LIN {X -109.277,Y -17.308,Z -54.438,A -90.000,B 90.000,C 0.000} C_DIS
LIN {X -109.528,Y -17.308,Z -53.967,A -90.000,B 90.000,C 0.000} C_DIS
LIN {X -109.760,Y -17.308,Z -53.459,A -90.000,B 90.000,C 0.000} C_DIS
LIN {X -109.870,Y -17.308,Z -53.202,A -90.000,B 90.000,C 0.000} C_DIS
LIN {X -109.990,Y -17.308,Z -52.935,A -90.000,B 90.000,C 0.000} C_DIS
LIN {X -110.022,Y -17.308,Z -52.850,A -90.000,B 90.000,C 0.000} C_DIS
LIN {X -110.260,Y -17.308,Z -52.116,A -90.000,B 90.000,C 0.000} C_DIS
LIN {X -110.354,Y -17.308,Z -51.704,A -90.000,B 90.000,C 0.000} C_DIS
LIN {X -110.399,Y -17.308,Z -51.283,A -90.000,B 90.000,C 0.000} C_DIS
LIN {X -110.450,Y -17.308,Z -50.683,A -90.000,B 90.000,C 0.000} C_DIS
LIN {X -110.444,Y -17.308,Z -50.213,A -90.000,B 90.000,C 0.000} C_DIS
LIN {X -110.434,Y -17.308,Z -50.113,A -90.000,B 90.000,C 0.000} C_DIS
LIN {X -110.392,Y -17.308,Z -49.798,A -90.000,B 90.000,C 0.000} C_DIS
LIN {X -110.361,Y -17.308,Z -49.609,A -90.000,B 90.000,C 0.000} C_DIS
LIN {X -110.302,Y -17.308,Z -49.301,A -90.000,B 90.000,C 0.000} C_DIS
LIN {X -110.171,Y -17.308,Z -48.794,A -90.000,B 90.000,C 0.000} C_DIS
LIN {X -110.038,Y -17.308,Z -48.429,A -90.000,B 90.000,C 0.000} C_DIS
LIN {X -109.863,Y -17.308,Z -47.985,A -90.000,B 90.000,C 0.000} C_DIS
LIN {X -109.731,Y -17.308,Z -47.725,A -90.000,B 90.000,C 0.000} C_DIS
LIN {X -109.686,Y -17.308,Z -47.627,A -90.000,B 90.000,C 0.000} C_DIS
LIN {X -109.488,Y -17.308,Z -47.252,A -90.000,B 90.000,C 0.000} C_DIS
LIN {X -109.413,Y -17.308,Z -47.127,A -90.000,B 90.000,C 0.000} C_DIS
LIN {X -109.830,Y -17.308,Z -46.394,A -90.000,B 90.000,C 0.000} C_DIS
LIN {X -109.928,Y -17.308,Z -46.209,A -90.000,B 90.000,C 0.000} C_DIS
LIN {X -110.117,Y -17.308,Z -45.841,A -90.000,B 90.000,C 0.000} C_DIS
LIN {X -110.455,Y -17.308,Z -45.092,A -90.000,B 90.000,C 0.000} C_DIS
LIN {X -110.509,Y -17.308,Z -44.961,A -90.000,B 90.000,C 0.000} C_DIS
LIN {X -110.701,Y -17.308,Z -44.445,A -90.000,B 90.000,C 0.000} C_DIS
LIN {X -110.791,Y -17.308,Z -44.174,A -90.000,B 90.000,C 0.000} C_DIS
LIN {X -110.988,Y -17.308,Z -43.576,A -90.000,B 90.000,C 0.000} C_DIS
LIN {X -111.093,Y -17.308,Z -43.162,A -90.000,B 90.000,C 0.000} C_DIS
LIN {X -111.179,Y -17.308,Z -42.781,A -90.000,B 90.000,C 0.000} C_DIS
LIN {X -111.225,Y -17.308,Z -42.559,A -90.000,B 90.000,C 0.000} C_DIS
LIN {X -111.305,Y -17.308,Z -42.009,A -90.000,B 90.000,C 0.000} C_DIS
LIN {X -111.349,Y -17.308,Z -41.588,A -90.000,B 90.000,C 0.000} C_DIS
LIN {X -111.368,Y -17.308,Z -41.241,A -90.000,B 90.000,C 0.000} C_DIS
LIN {X -111.364,Y -17.308,Z -40.978,A -90.000,B 90.000,C 0.000} C_DIS
LIN {X -111.359,Y -17.308,Z -40.623,A -90.000,B 90.000,C 0.000} C_DIS
LIN {X -111.346,Y -17.308,Z -40.304,A -90.000,B 90.000,C 0.000} C_DIS
LIN {X -111.305,Y -17.308,Z -39.903,A -90.000,B 90.000,C 0.000} C_DIS
LIN {X -111.262,Y -17.308,Z -39.606,A -90.000,B 90.000,C 0.000} C_DIS
LIN {X -111.171,Y -17.308,Z -39.214,A -90.000,B 90.000,C 0.000} C_DIS
LIN {X -111.102,Y -17.308,Z -38.934,A -90.000,B 90.000,C 0.000} C_DIS
LIN {X -110.936,Y -17.308,Z -38.436,A -90.000,B 90.000,C 0.000} C_DIS
LIN {X -110.874,Y -17.308,Z -38.268,A -90.000,B 90.000,C 0.000} C_DIS
LIN {X -110.765,Y -17.308,Z -38.003,A -90.000,B 90.000,C 0.000} C_DIS
LIN {X -110.667,Y -17.308,Z -37.794,A -90.000,B 90.000,C 0.000} C_DIS
LIN {X -110.600,Y -17.308,Z -37.663,A -90.000,B 90.000,C 0.000} C_DIS
LIN {X -110.459,Y -17.308,Z -37.399,A -90.000,B 90.000,C 0.000} C_DIS
LIN {X -110.237,Y -17.308,Z -37.056,A -90.000,B 90.000,C 0.000} C_DIS
LIN {X -110.078,Y -17.308,Z -36.846,A -90.000,B 90.000,C 0.000} C_DIS
LIN {X -109.834,Y -17.308,Z -36.557,A -90.000,B 90.000,C 0.000} C_DIS
LIN {X -109.557,Y -17.308,Z -36.304,A -90.000,B 90.000,C 0.000} C_DIS
LIN {X -109.328,Y -17.308,Z -36.101,A -90.000,B 90.000,C 0.000} C_DIS
LIN {X -109.011,Y -17.308,Z -35.882,A -90.000,B 90.000,C 0.000} C_DIS
LIN {X -108.744,Y -17.308,Z -35.735,A -90.000,B 90.000,C 0.000} C_DIS
LIN {X -108.407,Y -17.308,Z -35.562,A -90.000,B 90.000,C 0.000} C_DIS
LIN {X -108.370,Y -17.308,Z -35.547,A -90.000,B 90.000,C 0.000} C_DIS
LIN {X -108.101,Y -17.308,Z -35.424,A -90.000,B 90.000,C 0.000} C_DIS
LIN {X -108.024,Y -17.308,Z -35.397,A -90.000,B 90.000,C 0.000} C_DIS
LIN {X -107.986,Y -17.308,Z -35.382,A -90.000,B 90.000,C 0.000} C_DIS
LIN {X -107.790,Y -17.308,Z -35.138,A -90.000,B 90.000,C 0.000} C_DIS
LIN {X -107.687,Y -17.308,Z -35.003,A -90.000,B 90.000,C 0.000} C_DIS
LIN {X -107.576,Y -17.308,Z -34.852,A -90.000,B 90.000,C 0.000} C_DIS
LIN {X -107.363,Y -17.308,Z -34.573,A -90.000,B 90.000,C 0.000} C_DIS
LIN {X -107.172,Y -17.308,Z -34.351,A -90.000,B 90.000,C 0.000} C_DIS
LIN {X -106.994,Y -17.308,Z -34.130,A -90.000,B 90.000,C 0.000} C_DIS
LIN {X -106.743,Y -17.308,Z -33.884,A -90.000,B 90.000,C 0.000} C_DIS
LIN {X -106.465,Y -17.308,Z -33.618,A -90.000,B 90.000,C 0.000} C_DIS
LIN {X -106.295,Y -17.308,Z -33.457,A -90.000,B 90.000,C 0.000} C_DIS
LIN {X -105.896,Y -17.308,Z -33.133,A -90.000,B 90.000,C 0.000} C_DIS
LIN {X -105.714,Y -17.308,Z -32.987,A -90.000,B 90.000,C 0.000} C_DIS
LIN {X -104.978,Y -17.308,Z -32.450,A -90.000,B 90.000,C 0.000} C_DIS
LIN {X -104.425,Y -17.308,Z -32.079,A -90.000,B 90.000,C 0.000} C_DIS
LIN {X -104.048,Y -17.308,Z -31.825,A -90.000,B 90.000,C 0.000} C_DIS
LIN {X -103.908,Y -17.308,Z -31.733,A -90.000,B 90.000,C 0.000} C_DIS
LIN {X -103.388,Y -17.308,Z -31.409,A -90.000,B 90.000,C 0.000} C_DIS
LIN {X -102.835,Y -17.308,Z -31.110,A -90.000,B 90.000,C 0.000} C_DIS
LIN {X -102.526,Y -17.308,Z -30.944,A -90.000,B 90.000,C 0.000} C_DIS
LIN {X -102.329,Y -17.308,Z -30.848,A -90.000,B 90.000,C 0.000} C_DIS
LIN {X -101.877,Y -17.308,Z -30.649,A -90.000,B 90.000,C 0.000} C_DIS
LIN {X -101.633,Y -17.308,Z -30.551,A -90.000,B 90.000,C 0.000} C_DIS
LIN {X -101.290,Y -17.308,Z -30.421,A -90.000,B 90.000,C 0.000} C_DIS
LIN {X -100.896,Y -17.308,Z -30.282,A -90.000,B 90.000,C 0.000} C_DIS
LIN {X -100.530,Y -17.308,Z -30.139,A -90.000,B 90.000,C 0.000} C_DIS
LIN {X -100.458,Y -17.308,Z -29.896,A -90.000,B 90.000,C 0.000} C_DIS
LIN {X -100.322,Y -17.308,Z -29.499,A -90.000,B 90.000,C 0.000} C_DIS
LIN {X -100.161,Y -17.308,Z -29.156,A -90.000,B 90.000,C 0.000} C_DIS
LIN {X -99.930,Y -17.308,Z -28.698,A -90.000,B 90.000,C 0.000} C_DIS
LIN {X -99.695,Y -17.308,Z -28.324,A -90.000,B 90.000,C 0.000} C_DIS
LIN {X -99.528,Y -17.308,Z -28.064,A -90.000,B 90.000,C 0.000} C_DIS
LIN {X -99.432,Y -17.308,Z -27.919,A -90.000,B 90.000,C 0.000} C_DIS
LIN {X -99.092,Y -17.308,Z -27.475,A -90.000,B 90.000,C 0.000} C_DIS
LIN {X -98.825,Y -17.308,Z -27.155,A -90.000,B 90.000,C 0.000} C_DIS
LIN {X -98.539,Y -17.308,Z -26.819,A -90.000,B 90.000,C 0.000} C_DIS
LIN {X -98.265,Y -17.308,Z -26.515,A -90.000,B 90.000,C 0.000} C_DIS
LIN {X -98.055,Y -17.308,Z -26.298,A -90.000,B 90.000,C 0.000} C_DIS
LIN {X -97.848,Y -17.308,Z -26.093,A -90.000,B 90.000,C 0.000} C_DIS
LIN {X -97.651,Y -17.308,Z -25.907,A -90.000,B 90.000,C 0.000} C_DIS
LIN {X -97.470,Y -17.308,Z -25.741,A -90.000,B 90.000,C 0.000} C_DIS
LIN {X -97.372,Y -17.308,Z -25.646,A -90.000,B 90.000,C 0.000} C_DIS
LIN {X -97.070,Y -17.308,Z -25.379,A -90.000,B 90.000,C 0.000} C_DIS
LIN {X -96.977,Y -17.308,Z -25.311,A -90.000,B 90.000,C 0.000} C_DIS
LIN {X -96.877,Y -17.308,Z -25.234,A -90.000,B 90.000,C 0.000} C_DIS
LIN {X -96.544,Y -17.308,Z -25.007,A -90.000,B 90.000,C 0.000} C_DIS
LIN {X -96.186,Y -17.308,Z -24.822,A -90.000,B 90.000,C 0.000} C_DIS
LIN {X -95.601,Y -17.308,Z -24.606,A -90.000,B 90.000,C 0.000} C_DIS
LIN {X -95.394,Y -17.308,Z -24.551,A -90.000,B 90.000,C 0.000} C_DIS
LIN {X -95.167,Y -17.308,Z -24.498,A -90.000,B 90.000,C 0.000} C_DIS
LIN {X -95.084,Y -17.308,Z -24.484,A -90.000,B 90.000,C 0.000} C_DIS
LIN {X -94.665,Y -17.308,Z -24.424,A -90.000,B 90.000,C 0.000} C_DIS
LIN {X -94.242,Y -17.308,Z -24.415,A -90.000,B 90.000,C 0.000} C_DIS
LIN {X -94.028,Y -17.308,Z -24.425,A -90.000,B 90.000,C 0.000} C_DIS
LIN {X -93.391,Y -17.308,Z -24.450,A -90.000,B 90.000,C 0.000} C_DIS
LIN {X -93.076,Y -17.308,Z -24.495,A -90.000,B 90.000,C 0.000} C_DIS
LIN {X -92.696,Y -17.308,Z -24.538,A -90.000,B 90.000,C 0.000} C_DIS
LIN {X -92.367,Y -17.308,Z -24.604,A -90.000,B 90.000,C 0.000} C_DIS
LIN {X -92.079,Y -17.308,Z -24.636,A -90.000,B 90.000,C 0.000} C_DIS
LIN {X -91.937,Y -17.308,Z -24.654,A -90.000,B 90.000,C 0.000} C_DIS
LIN {X -91.341,Y -17.308,Z -24.709,A -90.000,B 90.000,C 0.000} C_DIS
LIN {X -90.954,Y -17.308,Z -24.728,A -90.000,B 90.000,C 0.000} C_DIS
LIN {X -90.765,Y -17.308,Z -24.739,A -90.000,B 90.000,C 0.000} C_DIS
LIN {X -90.252,Y -17.308,Z -24.737,A -90.000,B 90.000,C 0.000} C_DIS
LIN {X -89.583,Y -17.308,Z -24.703,A -90.000,B 90.000,C 0.000} C_DIS
LIN {X -89.336,Y -17.308,Z -24.674,A -90.000,B 90.000,C 0.000} C_DIS
LIN {X -88.613,Y -17.308,Z -24.546,A -90.000,B 90.000,C 0.000} C_DIS
LIN {X -88.432,Y -17.308,Z -24.502,A -90.000,B 90.000,C 0.000} C_DIS
LIN {X -88.062,Y -17.308,Z -24.386,A -90.000,B 90.000,C 0.000} C_DIS
LIN {X -87.996,Y -17.308,Z -24.360,A -90.000,B 90.000,C 0.000} C_DIS
LIN {X -87.766,Y -17.308,Z -24.270,A -90.000,B 90.000,C 0.000} C_DIS
LIN {X -87.464,Y -17.308,Z -24.122,A -90.000,B 90.000,C 0.000} C_DIS
LIN {X -87.249,Y -17.308,Z -23.989,A -90.000,B 90.000,C 0.000} C_DIS
LIN {X -87.134,Y -17.308,Z -23.898,A -90.000,B 90.000,C 0.000} C_DIS
LIN {X -87.088,Y -17.308,Z -23.852,A -90.000,B 90.000,C 0.000} C_DIS
LIN {X -86.793,Y -17.308,Z -23.483,A -90.000,B 90.000,C 0.000} C_DIS
LIN {X -86.245,Y -17.308,Z -22.709,A -90.000,B 90.000,C 0.000} C_DIS
LIN {X -85.958,Y -17.308,Z -22.315,A -90.000,B 90.000,C 0.000} C_DIS
LIN {X -85.762,Y -17.308,Z -22.052,A -90.000,B 90.000,C 0.000} C_DIS
LIN {X -85.514,Y -17.308,Z -21.715,A -90.000,B 90.000,C 0.000} C_DIS
LIN {X -85.447,Y -17.308,Z -21.614,A -90.000,B 90.000,C 0.000} C_DIS
LIN {X -85.429,Y -17.308,Z -21.548,A -90.000,B 90.000,C 0.000} C_DIS
LIN {X -85.386,Y -17.308,Z -21.370,A -90.000,B 90.000,C 0.000} C_DIS
LIN {X -85.352,Y -17.308,Z -21.224,A -90.000,B 90.000,C 0.000} C_DIS
LIN {X -85.295,Y -17.308,Z -21.008,A -90.000,B 90.000,C 0.000} C_DIS
LIN {X -85.173,Y -17.308,Z -20.564,A -90.000,B 90.000,C 0.000} C_DIS
LIN {X -85.006,Y -17.308,Z -20.118,A -90.000,B 90.000,C 0.000} C_DIS
LIN {X -84.875,Y -17.308,Z -19.788,A -90.000,B 90.000,C 0.000} C_DIS
LIN {X -84.669,Y -17.308,Z -19.377,A -90.000,B 90.000,C 0.000} C_DIS
LIN {X -84.438,Y -17.308,Z -18.974,A -90.000,B 90.000,C 0.000} C_DIS
LIN {X -84.069,Y -17.308,Z -18.464,A -90.000,B 90.000,C 0.000} C_DIS
LIN {X -83.972,Y -17.308,Z -18.336,A -90.000,B 90.000,C 0.000} C_DIS
LIN {X -83.659,Y -17.308,Z -17.989,A -90.000,B 90.000,C 0.000} C_DIS
LIN {X -83.310,Y -17.308,Z -17.678,A -90.000,B 90.000,C 0.000} C_DIS
LIN {X -83.039,Y -17.308,Z -17.445,A -90.000,B 90.000,C 0.000} C_DIS
LIN {X -82.804,Y -17.308,Z -17.264,A -90.000,B 90.000,C 0.000} C_DIS
LIN {X -82.421,Y -17.308,Z -17.018,A -90.000,B 90.000,C 0.000} C_DIS
LIN {X -82.064,Y -17.308,Z -16.803,A -90.000,B 90.000,C 0.000} C_DIS
LIN {X -81.656,Y -17.308,Z -16.601,A -90.000,B 90.000,C 0.000} C_DIS
LIN {X -81.272,Y -17.308,Z -16.447,A -90.000,B 90.000,C 0.000} C_DIS
LIN {X -80.773,Y -17.308,Z -16.264,A -90.000,B 90.000,C 0.000} C_DIS
LIN {X -80.331,Y -17.308,Z -16.156,A -90.000,B 90.000,C 0.000} C_DIS
LIN {X -79.940,Y -17.308,Z -16.064,A -90.000,B 90.000,C 0.000} C_DIS
LIN {X -79.763,Y -17.308,Z -16.028,A -90.000,B 90.000,C 0.000} C_DIS
LIN {X -79.312,Y -17.308,Z -15.968,A -90.000,B 90.000,C 0.000} C_DIS
LIN {X -78.986,Y -17.308,Z -15.938,A -90.000,B 90.000,C 0.000} C_DIS
LIN {X -78.616,Y -17.308,Z -15.911,A -90.000,B 90.000,C 0.000} C_DIS
LIN {X -78.161,Y -17.308,Z -15.902,A -90.000,B 90.000,C 0.000} C_DIS
LIN {X -77.499,Y -17.308,Z -15.925,A -90.000,B 90.000,C 0.000} C_DIS
LIN {X -77.301,Y -17.308,Z -15.936,A -90.000,B 90.000,C 0.000} C_DIS
LIN {X -76.909,Y -17.308,Z -15.971,A -90.000,B 90.000,C 0.000} C_DIS
LIN {X -76.875,Y -17.308,Z -15.976,A -90.000,B 90.000,C 0.000} C_DIS
LIN {X -75.728,Y -17.308,Z -16.188,A -90.000,B 90.000,C 0.000} C_DIS
LIN {X -75.480,Y -17.308,Z -16.245,A -90.000,B 90.000,C 0.000} C_DIS
LIN {X -74.439,Y -17.308,Z -16.560,A -90.000,B 90.000,C 0.000} C_DIS
LIN {X -73.971,Y -17.308,Z -16.709,A -90.000,B 90.000,C 0.000} C_DIS
LIN {X -72.559,Y -17.308,Z -17.306,A -90.000,B 90.000,C 0.000} C_DIS
LIN {X -72.171,Y -17.308,Z -17.515,A -90.000,B 90.000,C 0.000} C_DIS
LIN {X -71.532,Y -17.308,Z -17.863,A -90.000,B 90.000,C 0.000} C_DIS
LIN {X -71.248,Y -17.308,Z -18.011,A -90.000,B 90.000,C 0.000} C_DIS
LIN {X -70.853,Y -17.308,Z -18.223,A -90.000,B 90.000,C 0.000} C_DIS
LIN {X -70.304,Y -17.308,Z -18.552,A -90.000,B 90.000,C 0.000} C_DIS
LIN {X -69.506,Y -17.308,Z -19.020,A -90.000,B 90.000,C 0.000} C_DIS
LIN {X -69.055,Y -17.308,Z -19.311,A -90.000,B 90.000,C 0.000} C_DIS
LIN {X -67.940,Y -17.308,Z -20.084,A -90.000,B 90.000,C 0.000} C_DIS
LIN {X -67.668,Y -17.308,Z -20.290,A -90.000,B 90.000,C 0.000} C_DIS
LIN {X -67.045,Y -17.308,Z -20.777,A -90.000,B 90.000,C 0.000} C_DIS
LIN {X -66.717,Y -17.308,Z -21.045,A -90.000,B 90.000,C 0.000} C_DIS
LIN {X -66.444,Y -17.308,Z -21.276,A -90.000,B 90.000,C 0.000} C_DIS
LIN {X -65.961,Y -17.308,Z -21.696,A -90.000,B 90.000,C 0.000} C_DIS
LIN {X -65.767,Y -17.308,Z -21.893,A -90.000,B 90.000,C 0.000} C_DIS
LIN {X -65.312,Y -17.308,Z -22.358,A -90.000,B 90.000,C 0.000} C_DIS
LIN {X -64.845,Y -17.308,Z -22.810,A -90.000,B 90.000,C 0.000} C_DIS
LIN {X -64.258,Y -17.308,Z -23.509,A -90.000,B 90.000,C 0.000} C_DIS
LIN {X -63.904,Y -17.308,Z -23.932,A -90.000,B 90.000,C 0.000} C_DIS
LIN {X -63.462,Y -17.308,Z -24.494,A -90.000,B 90.000,C 0.000} C_DIS
LIN {X -63.348,Y -17.308,Z -24.652,A -90.000,B 90.000,C 0.000} C_DIS
LIN {X -63.215,Y -17.308,Z -24.848,A -90.000,B 90.000,C 0.000} C_DIS
LIN {X -62.785,Y -17.308,Z -25.397,A -90.000,B 90.000,C 0.000} C_DIS
LIN {X -62.557,Y -17.308,Z -25.702,A -90.000,B 90.000,C 0.000} C_DIS
LIN {X -62.483,Y -17.308,Z -25.777,A -90.000,B 90.000,C 0.000} C_DIS
LIN {X -62.054,Y -17.308,Z -26.201,A -90.000,B 90.000,C 0.000} C_DIS
LIN {X -61.340,Y -17.308,Z -26.673,A -90.000,B 90.000,C 0.000} C_DIS
LIN {X -60.531,Y -17.308,Z -27.025,A -90.000,B 90.000,C 0.000} C_DIS
LIN {X -60.319,Y -17.308,Z -27.118,A -90.000,B 90.000,C 0.000} C_DIS
LIN {X -58.849,Y -17.308,Z -27.587,A -90.000,B 90.000,C 0.000} C_DIS
LIN {X -56.852,Y -17.308,Z -28.118,A -90.000,B 90.000,C 0.000} C_DIS
LIN {X -56.644,Y -17.308,Z -28.164,A -90.000,B 90.000,C 0.000} C_DIS
LIN {X -55.206,Y -17.308,Z -28.534,A -90.000,B 90.000,C 0.000} C_DIS
LIN {X -54.599,Y -17.308,Z -28.678,A -90.000,B 90.000,C 0.000} C_DIS
LIN {X -53.961,Y -17.308,Z -28.823,A -90.000,B 90.000,C 0.000} C_DIS
LIN {X -52.713,Y -17.308,Z -29.052,A -90.000,B 90.000,C 0.000} C_DIS
LIN {X -52.238,Y -17.308,Z -29.158,A -90.000,B 90.000,C 0.000} C_DIS
LIN {X -50.712,Y -17.308,Z -29.450,A -90.000,B 90.000,C 0.000} C_DIS
LIN {X -49.140,Y -17.308,Z -29.676,A -90.000,B 90.000,C 0.000} C_DIS
LIN {X -48.828,Y -17.308,Z -29.708,A -90.000,B 90.000,C 0.000} C_DIS
LIN {X -45.658,Y -17.308,Z -30.077,A -90.000,B 90.000,C 0.000} C_DIS
LIN {X -45.116,Y -17.308,Z -30.119,A -90.000,B 90.000,C 0.000} C_DIS
LIN {X -44.038,Y -17.308,Z -30.215,A -90.000,B 90.000,C 0.000} C_DIS
LIN {X -41.956,Y -17.308,Z -30.414,A -90.000,B 90.000,C 0.000} C_DIS
LIN {X -40.163,Y -17.308,Z -30.556,A -90.000,B 90.000,C 0.000} C_DIS
LIN {X -39.196,Y -17.308,Z -30.672,A -90.000,B 90.000,C 0.000} C_DIS
LIN {X -36.171,Y -17.308,Z -31.051,A -90.000,B 90.000,C 0.000} C_DIS
LIN {X -34.413,Y -17.308,Z -31.305,A -90.000,B 90.000,C 0.000} C_DIS
LIN {X -31.571,Y -17.308,Z -31.816,A -90.000,B 90.000,C 0.000} C_DIS
LIN {X -29.817,Y -17.308,Z -32.125,A -90.000,B 90.000,C 0.000} C_DIS
LIN {X -29.213,Y -17.308,Z -32.239,A -90.000,B 90.000,C 0.000} C_DIS
LIN {X -28.110,Y -17.308,Z -32.443,A -90.000,B 90.000,C 0.000} C_DIS
LIN {X -27.159,Y -17.308,Z -32.634,A -90.000,B 90.000,C 0.000} C_DIS
LIN {X -26.260,Y -17.308,Z -32.801,A -90.000,B 90.000,C 0.000} C_DIS
LIN {X -25.100,Y -17.308,Z -33.024,A -90.000,B 90.000,C 0.000} C_DIS
LIN {X -23.949,Y -17.308,Z -33.230,A -90.000,B 90.000,C 0.000} C_DIS
LIN {X -22.934,Y -17.308,Z -33.425,A -90.000,B 90.000,C 0.000} C_DIS
LIN {X -20.611,Y -17.308,Z -33.882,A -90.000,B 90.000,C 0.000} C_DIS
LIN {X -20.347,Y -17.308,Z -33.940,A -90.000,B 90.000,C 0.000} C_DIS
LIN {X -19.518,Y -17.308,Z -34.105,A -90.000,B 90.000,C 0.000} C_DIS
LIN {X -18.829,Y -17.308,Z -34.238,A -90.000,B 90.000,C 0.000} C_DIS
LIN {X -17.988,Y -17.308,Z -34.379,A -90.000,B 90.000,C 0.000} C_DIS
LIN {X -16.209,Y -17.308,Z -34.745,A -90.000,B 90.000,C 0.000} C_DIS
LIN {X -15.578,Y -17.308,Z -34.859,A -90.000,B 90.000,C 0.000} C_DIS
LIN {X -15.219,Y -17.308,Z -34.927,A -90.000,B 90.000,C 0.000} C_DIS
LIN {X -14.772,Y -17.308,Z -35.030,A -90.000,B 90.000,C 0.000} C_DIS
LIN {X -12.936,Y -17.308,Z -35.395,A -90.000,B 90.000,C 0.000} C_DIS
LIN {X -12.591,Y -17.308,Z -35.447,A -90.000,B 90.000,C 0.000} C_DIS
LIN {X -11.559,Y -17.308,Z -35.638,A -90.000,B 90.000,C 0.000} C_DIS
LIN {X -10.386,Y -17.308,Z -35.821,A -90.000,B 90.000,C 0.000} C_DIS
LIN {X -9.911,Y -17.308,Z -35.909,A -90.000,B 90.000,C 0.000} C_DIS
LIN {X -9.565,Y -17.308,Z -35.959,A -90.000,B 90.000,C 0.000} C_DIS
LIN {X -8.147,Y -17.308,Z -36.207,A -90.000,B 90.000,C 0.000} C_DIS
LIN {X -6.600,Y -17.308,Z -36.402,A -90.000,B 90.000,C 0.000} C_DIS
LIN {X -6.373,Y -17.308,Z -36.436,A -90.000,B 90.000,C 0.000} C_DIS
LIN {X -5.975,Y -17.308,Z -36.475,A -90.000,B 90.000,C 0.000} C_DIS
LIN {X -4.287,Y -17.308,Z -36.746,A -90.000,B 90.000,C 0.000} C_DIS
LIN {X -3.747,Y -17.308,Z -36.810,A -90.000,B 90.000,C 0.000} C_DIS
LIN {X -2.105,Y -17.308,Z -36.981,A -90.000,B 90.000,C 0.000} C_DIS
LIN {X -1.067,Y -17.308,Z -37.105,A -90.000,B 90.000,C 0.000} C_DIS
LIN {X 0.535,Y -17.308,Z -37.243,A -90.000,B 90.000,C 0.000} C_DIS
LIN {X 2.482,Y -17.308,Z -37.445,A -90.000,B 90.000,C 0.000} C_DIS
LIN {X 4.011,Y -17.308,Z -37.649,A -90.000,B 90.000,C 0.000} C_DIS
LIN {X 4.508,Y -17.308,Z -37.725,A -90.000,B 90.000,C 0.000} C_DIS
LIN {X 6.518,Y -17.308,Z -38.010,A -90.000,B 90.000,C 0.000} C_DIS
LIN {X 7.495,Y -17.308,Z -38.195,A -90.000,B 90.000,C 0.000} C_DIS
LIN {X 9.210,Y -17.308,Z -38.474,A -90.000,B 90.000,C 0.000} C_DIS
LIN {X 10.152,Y -17.308,Z -38.666,A -90.000,B 90.000,C 0.000} C_DIS
LIN {X 11.680,Y -17.308,Z -38.921,A -90.000,B 90.000,C 0.000} C_DIS
LIN {X 13.109,Y -17.308,Z -39.193,A -90.000,B 90.000,C 0.000} C_DIS
LIN {X 13.984,Y -17.308,Z -39.328,A -90.000,B 90.000,C 0.000} C_DIS
LIN {X 15.976,Y -17.308,Z -39.600,A -90.000,B 90.000,C 0.000} C_DIS
LIN {X 16.409,Y -17.308,Z -39.652,A -90.000,B 90.000,C 0.000} C_DIS
LIN {X 17.396,Y -17.308,Z -39.693,A -90.000,B 90.000,C 0.000} C_DIS
LIN {X 19.409,Y -17.308,Z -39.659,A -90.000,B 90.000,C 0.000} C_DIS
LIN {X 20.175,Y -17.308,Z -39.617,A -90.000,B 90.000,C 0.000} C_DIS
LIN {X 21.776,Y -17.308,Z -39.482,A -90.000,B 90.000,C 0.000} C_DIS
LIN {X 23.521,Y -17.308,Z -39.307,A -90.000,B 90.000,C 0.000} C_DIS
LIN {X 24.002,Y -17.308,Z -39.264,A -90.000,B 90.000,C 0.000} C_DIS
LIN {X 25.329,Y -17.308,Z -39.131,A -90.000,B 90.000,C 0.000} C_DIS
LIN {X 25.924,Y -17.308,Z -39.045,A -90.000,B 90.000,C 0.000} C_DIS
LIN {X 26.439,Y -17.308,Z -38.976,A -90.000,B 90.000,C 0.000} C_DIS
LIN {X 27.087,Y -17.308,Z -38.911,A -90.000,B 90.000,C 0.000} C_DIS
LIN {X 27.304,Y -17.308,Z -38.873,A -90.000,B 90.000,C 0.000} C_DIS
LIN {X 27.723,Y -17.308,Z -38.813,A -90.000,B 90.000,C 0.000} C_DIS
LIN {X 28.516,Y -17.308,Z -38.720,A -90.000,B 90.000,C 0.000} C_DIS
LIN {X 29.009,Y -17.308,Z -38.669,A -90.000,B 90.000,C 0.000} C_DIS
LIN {X 29.052,Y -17.308,Z -38.666,A -90.000,B 90.000,C 0.000} C_DIS
LIN {X 29.117,Y -17.308,Z -38.655,A -90.000,B 90.000,C 0.000} C_DIS
LIN {X 29.423,Y -17.308,Z -38.615,A -90.000,B 90.000,C 0.000} C_DIS
LIN {X 30.450,Y -17.308,Z -38.492,A -90.000,B 90.000,C 0.000} C_DIS
LIN {X 30.849,Y -17.308,Z -38.463,A -90.000,B 90.000,C 0.000} C_DIS
LIN {X 31.235,Y -17.308,Z -38.446,A -90.000,B 90.000,C 0.000} C_DIS
LIN {X 31.826,Y -17.308,Z -38.371,A -90.000,B 90.000,C 0.000} C_DIS
LIN {X 32.386,Y -17.308,Z -38.306,A -90.000,B 90.000,C 0.000} C_DIS
LIN {X 33.525,Y -17.308,Z -38.260,A -90.000,B 90.000,C 0.000} C_DIS
LIN {X 33.823,Y -17.308,Z -38.223,A -90.000,B 90.000,C 0.000} C_DIS
LIN {X 34.402,Y -17.308,Z -38.180,A -90.000,B 90.000,C 0.000} C_DIS
LIN {X 35.483,Y -17.308,Z -38.143,A -90.000,B 90.000,C 0.000} C_DIS
LIN {X 36.492,Y -17.308,Z -38.136,A -90.000,B 90.000,C 0.000} C_DIS
LIN {X 36.756,Y -17.308,Z -38.139,A -90.000,B 90.000,C 0.000} C_DIS
LIN {X 38.001,Y -17.308,Z -38.196,A -90.000,B 90.000,C 0.000} C_DIS
LIN {X 39.626,Y -17.308,Z -38.309,A -90.000,B 90.000,C 0.000} C_DIS
LIN {X 42.353,Y -17.308,Z -38.731,A -90.000,B 90.000,C 0.000} C_DIS
LIN {X 42.529,Y -17.308,Z -38.756,A -90.000,B 90.000,C 0.000} C_DIS
LIN {X 43.036,Y -17.308,Z -38.849,A -90.000,B 90.000,C 0.000} C_DIS
LIN {X 44.117,Y -17.308,Z -39.121,A -90.000,B 90.000,C 0.000} C_DIS
LIN {X 45.216,Y -17.308,Z -39.444,A -90.000,B 90.000,C 0.000} C_DIS
LIN {X 45.800,Y -17.308,Z -39.618,A -90.000,B 90.000,C 0.000} C_DIS
LIN {X 46.387,Y -17.308,Z -39.804,A -90.000,B 90.000,C 0.000} C_DIS
LIN {X 48.320,Y -17.308,Z -40.607,A -90.000,B 90.000,C 0.000} C_DIS
LIN {X 49.467,Y -17.308,Z -41.106,A -90.000,B 90.000,C 0.000} C_DIS
LIN {X 49.658,Y -17.308,Z -41.202,A -90.000,B 90.000,C 0.000} C_DIS
LIN {X 52.060,Y -17.308,Z -42.475,A -90.000,B 90.000,C 0.000} C_DIS
LIN {X 52.489,Y -17.308,Z -42.707,A -90.000,B 90.000,C 0.000} C_DIS
LIN {X 52.699,Y -17.308,Z -42.823,A -90.000,B 90.000,C 0.000} C_DIS
LIN {X 55.104,Y -17.308,Z -44.340,A -90.000,B 90.000,C 0.000} C_DIS
LIN {X 55.508,Y -17.308,Z -44.614,A -90.000,B 90.000,C 0.000} C_DIS
LIN {X 57.720,Y -17.308,Z -46.256,A -90.000,B 90.000,C 0.000} C_DIS
LIN {X 60.057,Y -17.308,Z -48.231,A -90.000,B 90.000,C 0.000} C_DIS
LIN {X 61.120,Y -17.308,Z -49.128,A -90.000,B 90.000,C 0.000} C_DIS
LIN {X 61.640,Y -17.308,Z -49.550,A -90.000,B 90.000,C 0.000} C_DIS
LIN {X 62.363,Y -17.308,Z -50.087,A -90.000,B 90.000,C 0.000} C_DIS
LIN {X 63.432,Y -17.308,Z -50.888,A -90.000,B 90.000,C 0.000} C_DIS
LIN {X 63.508,Y -17.308,Z -50.948,A -90.000,B 90.000,C 0.000} C_DIS
LIN {X 63.832,Y -17.308,Z -51.158,A -90.000,B 90.000,C 0.000} C_DIS
LIN {X 65.197,Y -17.308,Z -52.044,A -90.000,B 90.000,C 0.000} C_DIS
LIN {X 65.647,Y -17.308,Z -52.313,A -90.000,B 90.000,C 0.000} C_DIS
LIN {X 66.715,Y -17.308,Z -52.915,A -90.000,B 90.000,C 0.000} C_DIS
LIN {X 67.246,Y -17.308,Z -53.218,A -90.000,B 90.000,C 0.000} C_DIS
LIN {X 67.457,Y -17.308,Z -53.333,A -90.000,B 90.000,C 0.000} C_DIS
LIN {X 68.958,Y -17.308,Z -54.182,A -90.000,B 90.000,C 0.000} C_DIS
LIN {X 69.732,Y -17.308,Z -54.615,A -90.000,B 90.000,C 0.000} C_DIS
LIN {X 71.933,Y -17.308,Z -55.925,A -90.000,B 90.000,C 0.000} C_DIS
LIN {X 73.961,Y -17.308,Z -57.259,A -90.000,B 90.000,C 0.000} C_DIS
LIN {X 74.363,Y -17.308,Z -57.526,A -90.000,B 90.000,C 0.000} C_DIS
LIN {X 74.519,Y -17.308,Z -57.648,A -90.000,B 90.000,C 0.000} C_DIS
LIN {X 76.117,Y -17.308,Z -58.869,A -90.000,B 90.000,C 0.000} C_DIS
LIN {X 76.474,Y -17.308,Z -59.164,A -90.000,B 90.000,C 0.000} C_DIS
LIN {X 77.810,Y -17.308,Z -60.341,A -90.000,B 90.000,C 0.000} C_DIS
LIN {X 77.946,Y -17.308,Z -60.458,A -90.000,B 90.000,C 0.000} C_DIS
LIN {X 78.708,Y -17.308,Z -61.103,A -90.000,B 90.000,C 0.000} C_DIS
LIN {X 78.726,Y -17.590,Z -61.118,A -90.000,B 90.000,C 0.000} C_DIS
LIN {X 78.762,Y -17.984,Z -61.147,A -90.000,B 90.000,C 0.000} C_DIS
LIN {X 78.797,Y -18.191,Z -61.177,A -90.000,B 90.000,C 0.000} C_DIS
LIN {X 78.831,Y -18.294,Z -61.205,A -90.000,B 90.000,C 0.000} C_DIS
LIN {X 78.899,Y -18.470,Z -61.261,A -90.000,B 90.000,C 0.000} C_DIS
LIN {X 79.028,Y -18.751,Z -61.366,A -90.000,B 90.000,C 0.000} C_DIS
LIN {X 79.150,Y -18.971,Z -61.463,A -90.000,B 90.000,C 0.000} C_DIS
LIN {X 79.264,Y -19.153,Z -61.552,A -90.000,B 90.000,C 0.000} C_DIS
LIN {X 79.371,Y -19.309,Z -61.633,A -90.000,B 90.000,C 0.000} C_DIS
LIN {X 79.608,Y -19.630,Z -61.803,A -90.000,B 90.000,C 0.000} C_DIS
LIN {X 79.640,Y -19.668,Z -61.824,A -90.000,B 90.000,C 0.000} C_DIS
LIN {X 79.646,Y -26.073,Z -61.828,A -90.000,B 90.000,C 0.000} C_DIS
LIN {X 79.651,Y -26.234,Z -61.831,A -90.000,B 90.000,C 0.000} C_DIS
LIN {X 79.692,Y -26.692,Z -61.858,A -90.000,B 90.000,C 0.000} C_DIS
LIN {X 79.732,Y -26.943,Z -61.882,A -90.000,B 90.000,C 0.000} C_DIS
LIN {X 79.806,Y -27.288,Z -61.926,A -90.000,B 90.000,C 0.000} C_DIS
LIN {X 79.875,Y -27.533,Z -61.962,A -90.000,B 90.000,C 0.000} C_DIS
LIN {X 79.908,Y -27.633,Z -61.977,A -90.000,B 90.000,C 0.000} C_DIS
LIN {X 79.969,Y -27.803,Z -62.002,A -90.000,B 90.000,C 0.000} C_DIS
LIN {X 80.024,Y -27.939,Z -62.020,A -90.000,B 90.000,C 0.000} C_DIS
LIN {X 80.075,Y -28.051,Z -62.031,A -90.000,B 90.000,C 0.000} C_DIS
LIN {X 80.122,Y -28.143,Z -62.035,A -90.000,B 90.000,C 0.000} C_DIS
LIN {X 80.164,Y -28.220,Z -62.033,A -90.000,B 90.000,C 0.000} C_DIS
LIN {X 80.184,Y -28.254,Z -62.029,A -90.000,B 90.000,C 0.000} C_DIS
LIN {X 80.220,Y -28.313,Z -62.016,A -90.000,B 90.000,C 0.000} C_DIS
LIN {X 80.253,Y -28.361,Z -61.996,A -90.000,B 90.000,C 0.000} C_DIS
LIN {X 80.268,Y -28.381,Z -61.984,A -90.000,B 90.000,C 0.000} C_DIS
LIN {X 80.295,Y -28.414,Z -61.954,A -90.000,B 90.000,C 0.000} C_DIS
LIN {X 80.320,Y -28.436,Z -61.918,A -90.000,B 90.000,C 0.000} C_DIS
LIN {X 80.331,Y -28.443,Z -61.897,A -90.000,B 90.000,C 0.000} C_DIS
LIN {X 80.352,Y -28.451,Z -61.852,A -90.000,B 90.000,C 0.000} C_DIS
LIN {X 80.370,Y -28.451,Z -61.799,A -90.000,B 90.000,C 0.000} C_DIS
LIN {X 80.386,Y -28.442,Z -61.741,A -90.000,B 90.000,C 0.000} C_DIS
LIN {X 80.401,Y -28.426,Z -61.677,A -90.000,B 90.000,C 0.000} C_DIS
LIN {X 80.413,Y -28.403,Z -61.606,A -90.000,B 90.000,C 0.000} C_DIS
LIN {X 80.435,Y -28.338,Z -61.448,A -90.000,B 90.000,C 0.000} C_DIS
LIN {X 80.453,Y -28.251,Z -61.266,A -90.000,B 90.000,C 0.000} C_DIS
LIN {X 80.470,Y -28.146,Z -61.061,A -90.000,B 90.000,C 0.000} C_DIS
LIN {X 80.487,Y -28.022,Z -60.835,A -90.000,B 90.000,C 0.000} C_DIS
LIN {X 80.508,Y -27.874,Z -60.587,A -90.000,B 90.000,C 0.000} C_DIS
LIN {X 80.533,Y -27.702,Z -60.318,A -90.000,B 90.000,C 0.000} C_DIS
LIN {X 80.548,Y -27.606,Z -60.176,A -90.000,B 90.000,C 0.000} C_DIS
LIN {X 80.565,Y -27.501,Z -60.030,A -90.000,B 90.000,C 0.000} C_DIS
LIN {X 80.584,Y -27.387,Z -59.878,A -90.000,B 90.000,C 0.000} C_DIS
LIN {X 80.630,Y -27.125,Z -59.561,A -90.000,B 90.000,C 0.000} C_DIS
LIN {X 80.657,Y -26.994,Z -59.395,A -90.000,B 90.000,C 0.000} C_DIS
LIN {X 80.722,Y -26.804,Z -59.050,A -90.000,B 90.000,C 0.000} C_DIS
LIN {X 80.760,Y -26.706,Z -58.871,A -90.000,B 90.000,C 0.000} C_DIS
LIN {X 80.802,Y -26.608,Z -58.688,A -90.000,B 90.000,C 0.000} C_DIS
LIN {X 80.848,Y -26.509,Z -58.500,A -90.000,B 90.000,C 0.000} C_DIS
LIN {X 80.899,Y -26.413,Z -58.309,A -90.000,B 90.000,C 0.000} C_DIS
LIN {X 80.954,Y -26.321,Z -58.113,A -90.000,B 90.000,C 0.000} C_DIS
LIN {X 81.015,Y -26.239,Z -57.913,A -90.000,B 90.000,C 0.000} C_DIS
LIN {X 81.081,Y -26.175,Z -57.710,A -90.000,B 90.000,C 0.000} C_DIS
LIN {X 81.115,Y -26.153,Z -57.607,A -90.000,B 90.000,C 0.000} C_DIS
LIN {X 81.152,Y -26.139,Z -57.503,A -90.000,B 90.000,C 0.000} C_DIS
LIN {X 81.190,Y -26.134,Z -57.397,A -90.000,B 90.000,C 0.000} C_DIS
LIN {X 81.229,Y -26.121,Z -57.292,A -90.000,B 90.000,C 0.000} C_DIS
LIN {X 81.270,Y -26.089,Z -57.185,A -90.000,B 90.000,C 0.000} C_DIS
LIN {X 81.356,Y -25.986,Z -56.968,A -90.000,B 90.000,C 0.000} C_DIS
LIN {X 81.402,Y -25.943,Z -56.859,A -90.000,B 90.000,C 0.000} C_DIS
LIN {X 81.449,Y -25.914,Z -56.748,A -90.000,B 90.000,C 0.000} C_DIS
LIN {X 81.498,Y -17.308,Z -56.637,A -90.000,B 90.000,C 0.000} C_DIS
LIN {X 81.700,Y -17.308,Z -56.182,A -90.000,B 90.000,C 0.000} C_DIS
LIN {X 82.134,Y -17.308,Z -55.110,A -90.000,B 90.000,C 0.000} C_DIS
LIN {X 82.335,Y -17.308,Z -54.666,A -90.000,B 90.000,C 0.000} C_DIS
LIN {X 83.331,Y -17.308,Z -52.811,A -90.000,B 90.000,C 0.000} C_DIS
LIN {X 83.577,Y -17.308,Z -52.389,A -90.000,B 90.000,C 0.000} C_DIS
LIN {X 84.737,Y -17.308,Z -50.685,A -90.000,B 90.000,C 0.000} C_DIS
LIN {X 85.025,Y -17.308,Z -50.291,A -90.000,B 90.000,C 0.000} C_DIS
LIN {X 86.337,Y -17.308,Z -48.714,A -90.000,B 90.000,C 0.000} C_DIS
LIN {X 86.664,Y -17.308,Z -48.352,A -90.000,B 90.000,C 0.000} C_DIS
LIN {X 88.117,Y -17.308,Z -46.880,A -90.000,B 90.000,C 0.000} C_DIS
LIN {X 88.455,Y -17.308,Z -46.574,A -90.000,B 90.000,C 0.000} C_DIS
LIN {X 90.061,Y -17.308,Z -45.164,A -90.000,B 90.000,C 0.000} C_DIS
LIN {X 91.716,Y -17.308,Z -43.876,A -90.000,B 90.000,C 0.000} C_DIS
LIN {X 92.110,Y -17.308,Z -43.588,A -90.000,B 90.000,C 0.000} C_DIS
LIN {X 93.780,Y -17.308,Z -42.419,A -90.000,B 90.000,C 0.000} C_DIS
LIN {X 95.417,Y -17.308,Z -41.383,A -90.000,B 90.000,C 0.000} C_DIS
LIN {X 95.838,Y -17.308,Z -41.136,A -90.000,B 90.000,C 0.000} C_DIS
LIN {X 97.376,Y -17.308,Z -40.260,A -90.000,B 90.000,C 0.000} C_DIS
LIN {X 98.805,Y -17.308,Z -39.523,A -90.000,B 90.000,C 0.000} C_DIS
LIN {X 100.266,Y -17.308,Z -38.830,A -90.000,B 90.000,C 0.000} C_DIS
LIN {X 100.425,Y -17.308,Z -38.758,A -90.000,B 90.000,C 0.000} C_DIS
LIN {X 102.038,Y -17.308,Z -38.027,A -90.000,B 90.000,C 0.000} C_DIS
LIN {X 103.228,Y -17.308,Z -37.495,A -90.000,B 90.000,C 0.000} C_DIS
LIN {X 104.475,Y -17.308,Z -36.943,A -90.000,B 90.000,C 0.000} C_DIS
LIN {X 105.369,Y -17.308,Z -36.566,A -90.000,B 90.000,C 0.000} C_DIS
LIN {X 106.844,Y -17.308,Z -35.979,A -90.000,B 90.000,C 0.000} C_DIS
LIN {X 107.371,Y -17.308,Z -35.778,A -90.000,B 90.000,C 0.000} C_DIS
LIN {X 107.855,Y -17.308,Z -35.604,A -90.000,B 90.000,C 0.000} C_DIS
LIN {X 108.317,Y -17.308,Z -35.448,A -90.000,B 90.000,C 0.000} C_DIS
LIN {X 108.745,Y -17.308,Z -35.333,A -90.000,B 90.000,C 0.000} C_DIS
LIN {X 109.221,Y -17.308,Z -35.225,A -90.000,B 90.000,C 0.000} C_DIS
LIN {X 109.624,Y -17.308,Z -35.172,A -90.000,B 90.000,C 0.000} C_DIS
LIN {X 110.108,Y -17.308,Z -35.113,A -90.000,B 90.000,C 0.000} C_DIS
LIN {X 110.596,Y -17.308,Z -35.105,A -90.000,B 90.000,C 0.000} C_DIS
LIN {X 110.949,Y -17.308,Z -35.117,A -90.000,B 90.000,C 0.000} C_DIS
LIN {X 111.435,Y -17.308,Z -35.158,A -90.000,B 90.000,C 0.000} C_DIS
LIN {X 112.068,Y -17.308,Z -35.277,A -90.000,B 90.000,C 0.000} C_DIS
LIN {X 112.405,Y -17.308,Z -35.362,A -90.000,B 90.000,C 0.000} C_DIS
LIN {X 112.872,Y -17.308,Z -35.502,A -90.000,B 90.000,C 0.000} C_DIS
LIN {X 113.055,Y -17.308,Z -35.560,A -90.000,B 90.000,C 0.000} C_DIS
LIN {X 113.505,Y -17.308,Z -35.746,A -90.000,B 90.000,C 0.000} C_DIS
LIN {X 113.979,Y -17.308,Z -35.973,A -90.000,B 90.000,C 0.000} C_DIS
LIN {X 114.409,Y -17.308,Z -36.204,A -90.000,B 90.000,C 0.000} C_DIS
LIN {X 114.540,Y -17.308,Z -36.286,A -90.000,B 90.000,C 0.000} C_DIS
LIN {X 114.944,Y -17.308,Z -36.560,A -90.000,B 90.000,C 0.000} C_DIS
LIN {X 115.050,Y -17.308,Z -36.644,A -90.000,B 90.000,C 0.000} C_DIS
LIN {X 115.423,Y -17.308,Z -36.958,A -90.000,B 90.000,C 0.000} C_DIS
LIN {X 115.513,Y -17.308,Z -37.039,A -90.000,B 90.000,C 0.000} C_DIS
LIN {X 115.852,Y -17.308,Z -37.389,A -90.000,B 90.000,C 0.000} C_DIS
LIN {X 116.075,Y -17.308,Z -37.626,A -90.000,B 90.000,C 0.000} C_DIS
LIN {X 116.257,Y -17.308,Z -37.856,A -90.000,B 90.000,C 0.000} C_DIS
LIN {X 116.439,Y -17.308,Z -38.088,A -90.000,B 90.000,C 0.000} C_DIS
LIN {X 116.700,Y -17.308,Z -38.500,A -90.000,B 90.000,C 0.000} C_DIS
LIN {X 116.917,Y -17.308,Z -38.937,A -90.000,B 90.000,C 0.000} C_DIS
LIN {X 117.056,Y -17.308,Z -39.243,A -90.000,B 90.000,C 0.000} C_DIS
LIN {X 117.074,Y -17.308,Z -39.286,A -90.000,B 90.000,C 0.000} C_DIS
LIN {X 117.260,Y -17.308,Z -39.781,A -90.000,B 90.000,C 0.000} C_DIS
LIN {X 117.384,Y -17.308,Z -40.253,A -90.000,B 90.000,C 0.000} C_DIS
LIN {X 117.462,Y -17.308,Z -40.593,A -90.000,B 90.000,C 0.000} C_DIS
LIN {X 117.526,Y -17.308,Z -41.012,A -90.000,B 90.000,C 0.000} C_DIS
LIN {X 117.593,Y -17.308,Z -41.494,A -90.000,B 90.000,C 0.000} C_DIS
LIN {X 117.630,Y -17.308,Z -41.874,A -90.000,B 90.000,C 0.000} C_DIS
LIN {X 117.655,Y -17.308,Z -42.361,A -90.000,B 90.000,C 0.000} C_DIS
LIN {X 117.668,Y -17.308,Z -42.685,A -90.000,B 90.000,C 0.000} C_DIS
LIN {X 117.665,Y -17.308,Z -42.838,A -90.000,B 90.000,C 0.000} C_DIS
LIN {X 117.651,Y -17.308,Z -43.202,A -90.000,B 90.000,C 0.000} C_DIS
LIN {X 117.616,Y -17.308,Z -43.625,A -90.000,B 90.000,C 0.000} C_DIS
LIN {X 117.567,Y -17.308,Z -44.117,A -90.000,B 90.000,C 0.000} C_DIS
LIN {X 117.489,Y -17.308,Z -44.635,A -90.000,B 90.000,C 0.000} C_DIS
LIN {X 117.399,Y -17.308,Z -45.114,A -90.000,B 90.000,C 0.000} C_DIS
LIN {X 117.260,Y -17.308,Z -45.739,A -90.000,B 90.000,C 0.000} C_DIS
LIN {X 117.188,Y -17.308,Z -45.982,A -90.000,B 90.000,C 0.000} C_DIS
LIN {X 116.900,Y -17.308,Z -46.938,A -90.000,B 90.000,C 0.000} C_DIS
LIN {X 116.558,Y -17.308,Z -47.827,A -90.000,B 90.000,C 0.000} C_DIS
LIN {X 116.372,Y -17.308,Z -48.278,A -90.000,B 90.000,C 0.000} C_DIS
LIN {X 115.873,Y -17.308,Z -49.350,A -90.000,B 90.000,C 0.000} C_DIS
LIN {X 115.280,Y -17.308,Z -50.537,A -90.000,B 90.000,C 0.000} C_DIS
LIN {X 114.622,Y -17.308,Z -51.838,A -90.000,B 90.000,C 0.000} C_DIS
LIN {X 113.941,Y -17.308,Z -53.229,A -90.000,B 90.000,C 0.000} C_DIS
LIN {X 113.276,Y -17.308,Z -54.687,A -90.000,B 90.000,C 0.000} C_DIS
LIN {X 113.104,Y -17.308,Z -55.100,A -90.000,B 90.000,C 0.000} C_DIS
LIN {X 113.109,Y -17.401,Z -55.123,A -90.000,B 90.000,C 0.000} C_DIS
LIN {X 112.708,Y -17.540,Z -56.073,A -90.000,B 90.000,C 0.000} C_DIS
LIN {X 112.707,Y -34.735,Z -56.077,A -90.000,B 90.000,C 0.000} C_DIS
LIN {X 112.702,Y -34.774,Z -56.088,A -90.000,B 90.000,C 0.000} C_DIS
LIN {X 112.696,Y -34.805,Z -56.102,A -90.000,B 90.000,C 0.000} C_DIS
LIN {X 112.685,Y -34.849,Z -56.130,A -90.000,B 90.000,C 0.000} C_DIS
LIN {X 112.638,Y -34.954,Z -56.239,A -90.000,B 90.000,C 0.000} C_DIS
LIN {X 112.593,Y -35.023,Z -56.344,A -90.000,B 90.000,C 0.000} C_DIS
LIN {X 112.507,Y -35.128,Z -56.543,A -90.000,B 90.000,C 0.000} C_DIS
LIN {X 112.353,Y -35.330,Z -56.898,A -90.000,B 90.000,C 0.000} C_DIS
LIN {X 112.220,Y -35.524,Z -57.197,A -90.000,B 90.000,C 0.000} C_DIS
LIN {X 112.108,Y -35.707,Z -57.446,A -90.000,B 90.000,C 0.000} C_DIS
LIN {X 112.014,Y -35.947,Z -57.650,A -90.000,B 90.000,C 0.000} C_DIS
LIN {X 111.938,Y -36.098,Z -57.812,A -90.000,B 90.000,C 0.000} C_DIS
LIN {X 111.831,Y -36.280,Z -58.028,A -90.000,B 90.000,C 0.000} C_DIS
LIN {X 111.795,Y -36.340,Z -58.093,A -90.000,B 90.000,C 0.000} C_DIS
LIN {X 111.770,Y -36.387,Z -58.135,A -90.000,B 90.000,C 0.000} C_DIS
LIN {X 111.743,Y -36.451,Z -58.173,A -90.000,B 90.000,C 0.000} C_DIS
LIN {X 111.738,Y -36.470,Z -58.177,A -90.000,B 90.000,C 0.000} C_DIS
LIN {X 111.749,Y -36.397,Z -58.190,A -90.000,B 90.000,C 0.000} C_DIS
LIN {X 111.753,Y -36.342,Z -58.210,A -90.000,B 90.000,C 0.000} C_DIS
LIN {X 111.755,Y -36.274,Z -58.245,A -90.000,B 90.000,C 0.000} C_DIS
LIN {X 111.753,Y -36.187,Z -58.300,A -90.000,B 90.000,C 0.000} C_DIS
LIN {X 111.745,Y -36.075,Z -58.378,A -90.000,B 90.000,C 0.000} C_DIS
LIN {X 111.729,Y -35.926,Z -58.486,A -90.000,B 90.000,C 0.000} C_DIS
LIN {X 111.668,Y -35.425,Z -58.803,A -90.000,B 90.000,C 0.000} C_DIS
LIN {X 111.620,Y -35.114,Z -59.023,A -90.000,B 90.000,C 0.000} C_DIS
LIN {X 111.559,Y -34.895,Z -59.289,A -90.000,B 90.000,C 0.000} C_DIS
LIN {X 111.482,Y -34.695,Z -59.608,A -90.000,B 90.000,C 0.000} C_DIS
LIN {X 111.388,Y -34.464,Z -59.983,A -90.000,B 90.000,C 0.000} C_DIS
LIN {X 111.334,Y -34.295,Z -60.193,A -90.000,B 90.000,C 0.000} C_DIS
LIN {X 111.320,Y -34.228,Z -60.248,A -90.000,B 90.000,C 0.000} C_DIS
LIN {X 111.313,Y -34.176,Z -60.276,A -90.000,B 90.000,C 0.000} C_DIS
LIN {X 111.310,Y -34.135,Z -60.286,A -90.000,B 90.000,C 0.000} C_DIS
LIN {X 111.310,Y -17.604,Z -60.288,A -90.000,B 90.000,C 0.000} C_DIS
LIN {X 111.143,Y -17.541,Z -60.921,A -90.000,B 90.000,C 0.000} C_DIS
LIN {X 110.994,Y -17.499,Z -61.475,A -90.000,B 90.000,C 0.000} C_DIS
LIN {X 110.975,Y -17.308,Z -61.490,A -90.000,B 90.000,C 0.000} C_DIS
LIN {X 110.736,Y -17.308,Z -62.369,A -90.000,B 90.000,C 0.000} C_DIS
LIN {X 110.160,Y -17.308,Z -64.411,A -90.000,B 90.000,C 0.000} C_DIS
LIN {X 110.021,Y -17.308,Z -64.879,A -90.000,B 90.000,C 0.000} C_DIS
LIN {X 109.345,Y -17.308,Z -67.050,A -90.000,B 90.000,C 0.000} C_DIS
LIN {X 108.519,Y -17.308,Z -69.358,A -90.000,B 90.000,C 0.000} C_DIS
LIN {X 107.589,Y -17.308,Z -71.699,A -90.000,B 90.000,C 0.000} C_DIS
LIN {X 107.403,Y -17.308,Z -72.150,A -90.000,B 90.000,C 0.000} C_DIS
LIN {X 106.414,Y -17.308,Z -74.420,A -90.000,B 90.000,C 0.000} C_DIS
LIN {X 105.411,Y -17.308,Z -76.516,A -90.000,B 90.000,C 0.000} C_DIS
LIN {X 104.230,Y -17.308,Z -78.723,A -90.000,B 90.000,C 0.000} C_DIS
LIN {X 103.987,Y -17.308,Z -79.149,A -90.000,B 90.000,C 0.000} C_DIS
LIN {X 103.058,Y -17.308,Z -80.726,A -90.000,B 90.000,C 0.000} C_DIS
LIN {X 102.198,Y -17.308,Z -82.078,A -90.000,B 90.000,C 0.000} C_DIS
LIN {X 99.737,Y -17.308,Z -85.762,A -90.000,B 90.000,C 0.000} C_DIS
LIN {X 99.858,Y -17.308,Z -87.310,A -90.000,B 90.000,C 0.000} C_DIS
LIN {X 100.041,Y -17.308,Z -89.919,A -90.000,B 90.000,C 0.000} C_DIS
LIN {X 100.045,Y -17.308,Z -89.957,A -90.000,B 90.000,C 0.000} C_DIS
LIN {X 100.055,Y -17.308,Z -89.995,A -90.000,B 90.000,C 0.000} C_DIS
LIN {X 100.230,Y -17.308,Z -90.520,A -90.000,B 90.000,C 0.000} C_DIS
LIN {X 100.336,Y -17.308,Z -90.805,A -90.000,B 90.000,C 0.000} C_DIS
LIN {X 100.669,Y -17.308,Z -91.754,A -90.000,B 90.000,C 0.000} C_DIS
LIN {X 100.792,Y -17.308,Z -92.224,A -90.000,B 90.000,C 0.000} C_DIS
LIN {X 100.884,Y -17.308,Z -92.617,A -90.000,B 90.000,C 0.000} C_DIS
LIN {X 100.979,Y -17.308,Z -92.944,A -90.000,B 90.000,C 0.000} C_DIS
LIN {X 101.103,Y -17.308,Z -93.414,A -90.000,B 90.000,C 0.000} C_DIS
LIN {X 101.169,Y -17.308,Z -93.839,A -90.000,B 90.000,C 0.000} C_DIS
LIN {X 101.324,Y -17.308,Z -94.594,A -90.000,B 90.000,C 0.000} C_DIS
LIN {X 101.403,Y -17.308,Z -95.091,A -90.000,B 90.000,C 0.000} C_DIS
LIN {X 101.420,Y -17.308,Z -95.278,A -90.000,B 90.000,C 0.000} C_DIS
LIN {X 101.558,Y -17.308,Z -96.201,A -90.000,B 90.000,C 0.000} C_DIS
LIN {X 101.569,Y -17.308,Z -96.362,A -90.000,B 90.000,C 0.000} C_DIS
LIN {X 101.691,Y -17.308,Z -97.320,A -90.000,B 90.000,C 0.000} C_DIS
LIN {X 101.704,Y -17.308,Z -97.402,A -90.000,B 90.000,C 0.000} C_DIS
LIN {X 101.844,Y -17.308,Z -98.388,A -90.000,B 90.000,C 0.000} C_DIS
LIN {X 101.877,Y -17.308,Z -98.647,A -90.000,B 90.000,C 0.000} C_DIS
LIN {X 102.084,Y -17.308,Z -100.015,A -90.000,B 90.000,C 0.000} C_DIS
LIN {X 102.091,Y -17.308,Z -100.091,A -90.000,B 90.000,C 0.000} C_DIS
LIN {X 102.314,Y -17.308,Z -101.517,A -90.000,B 90.000,C 0.000} C_DIS
LIN {X 102.330,Y -17.308,Z -101.686,A -90.000,B 90.000,C 0.000} C_DIS
LIN {X 102.338,Y -17.308,Z -101.733,A -90.000,B 90.000,C 0.000} C_DIS
LIN {X 102.466,Y -17.308,Z -102.563,A -90.000,B 90.000,C 0.000} C_DIS
LIN {X 102.592,Y -17.308,Z -103.367,A -90.000,B 90.000,C 0.000} C_DIS
LIN {X 102.653,Y -17.308,Z -103.784,A -90.000,B 90.000,C 0.000} C_DIS
LIN {X 102.972,Y -17.308,Z -105.812,A -90.000,B 90.000,C 0.000} C_DIS
LIN {X 103.123,Y -17.308,Z -106.801,A -90.000,B 90.000,C 0.000} C_DIS
LIN {X 103.432,Y -17.308,Z -108.888,A -90.000,B 90.000,C 0.000} C_DIS
LIN {X 103.476,Y -17.308,Z -109.197,A -90.000,B 90.000,C 0.000} C_DIS
LIN {X 103.701,Y -17.308,Z -110.845,A -90.000,B 90.000,C 0.000} C_DIS
LIN {X 103.798,Y -17.308,Z -111.569,A -90.000,B 90.000,C 0.000} C_DIS
LIN {X 104.104,Y -17.308,Z -114.022,A -90.000,B 90.000,C 0.000} C_DIS
LIN {X 104.242,Y -17.308,Z -115.285,A -90.000,B 90.000,C 0.000} C_DIS
LIN {X 104.387,Y -17.308,Z -116.529,A -90.000,B 90.000,C 0.000} C_DIS
LIN {X 104.462,Y -17.308,Z -117.307,A -90.000,B 90.000,C 0.000} C_DIS
LIN {X 104.652,Y -17.308,Z -119.079,A -90.000,B 90.000,C 0.000} C_DIS
LIN {X 104.875,Y -17.308,Z -121.404,A -90.000,B 90.000,C 0.000} C_DIS
LIN {X 104.896,Y -17.308,Z -121.602,A -90.000,B 90.000,C 0.000} C_DIS
LIN {X 105.065,Y -17.308,Z -123.644,A -90.000,B 90.000,C 0.000} C_DIS
LIN {X 105.106,Y -17.308,Z -124.099,A -90.000,B 90.000,C 0.000} C_DIS
LIN {X 105.271,Y -17.308,Z -126.535,A -90.000,B 90.000,C 0.000} C_DIS
LIN {X 105.296,Y -17.308,Z -127.010,A -90.000,B 90.000,C 0.000} C_DIS
LIN {X 105.408,Y -17.308,Z -129.495,A -90.000,B 90.000,C 0.000} C_DIS
LIN {X 105.422,Y -17.308,Z -130.303,A -90.000,B 90.000,C 0.000} C_DIS
LIN {X 105.462,Y -17.308,Z -132.138,A -90.000,B 90.000,C 0.000} C_DIS
LIN {X 105.456,Y -17.308,Z -133.137,A -90.000,B 90.000,C 0.000} C_DIS
LIN {X 105.454,Y -17.308,Z -135.049,A -90.000,B 90.000,C 0.000} C_DIS
LIN {X 105.411,Y -17.308,Z -137.048,A -90.000,B 90.000,C 0.000} C_DIS
LIN {X 105.379,Y -17.308,Z -138.366,A -90.000,B 90.000,C 0.000} C_DIS
LIN {X 105.258,Y -17.308,Z -141.622,A -90.000,B 90.000,C 0.000} C_DIS
LIN {X 105.232,Y -17.308,Z -142.272,A -90.000,B 90.000,C 0.000} C_DIS
LIN {X 105.041,Y -17.308,Z -146.025,A -90.000,B 90.000,C 0.000} C_DIS
LIN {X 104.798,Y -17.308,Z -149.863,A -90.000,B 90.000,C 0.000} C_DIS
LIN {X 104.508,Y -17.308,Z -153.692,A -90.000,B 90.000,C 0.000} C_DIS
LIN {X 104.183,Y -17.308,Z -157.492,A -90.000,B 90.000,C 0.000} C_DIS
LIN {X 103.833,Y -17.308,Z -161.241,A -90.000,B 90.000,C 0.000} C_DIS
LIN {X 103.473,Y -17.308,Z -164.912,A -90.000,B 90.000,C 0.000} C_DIS
LIN {X 103.061,Y -17.308,Z -169.022,A -90.000,B 90.000,C 0.000} C_DIS
LIN {X 102.758,Y -17.308,Z -171.927,A -90.000,B 90.000,C 0.000} C_DIS
LIN {X 102.397,Y -17.308,Z -175.185,A -90.000,B 90.000,C 0.000} C_DIS
LIN {X 102.028,Y -17.308,Z -178.226,A -90.000,B 90.000,C 0.000} C_DIS
LIN {X 101.779,Y -17.308,Z -180.058,A -90.000,B 90.000,C 0.000} C_DIS
LIN {X 101.643,Y -17.308,Z -181.040,A -90.000,B 90.000,C 0.000} C_DIS
LIN {X 101.579,Y -17.308,Z -181.481,A -90.000,B 90.000,C 0.000} C_DIS
LIN {X 101.189,Y -17.308,Z -184.066,A -90.000,B 90.000,C 0.000} C_DIS
LIN {X 100.422,Y -17.308,Z -188.908,A -90.000,B 90.000,C 0.000} C_DIS
LIN {X 100.058,Y -17.308,Z -191.287,A -90.000,B 90.000,C 0.000} C_DIS
LIN {X 99.634,Y -17.308,Z -193.944,A -90.000,B 90.000,C 0.000} C_DIS
LIN {X 99.477,Y -17.308,Z -194.890,A -90.000,B 90.000,C 0.000} C_DIS
LIN {X 99.119,Y -17.308,Z -196.914,A -90.000,B 90.000,C 0.000} C_DIS
LIN {X 98.882,Y -17.308,Z -198.230,A -90.000,B 90.000,C 0.000} C_DIS
LIN {X 98.444,Y -17.308,Z -200.459,A -90.000,B 90.000,C 0.000} C_DIS
LIN {X 98.089,Y -17.308,Z -202.279,A -90.000,B 90.000,C 0.000} C_DIS
LIN {X 97.552,Y -17.308,Z -204.773,A -90.000,B 90.000,C 0.000} C_DIS
LIN {X 97.074,Y -17.308,Z -207.076,A -90.000,B 90.000,C 0.000} C_DIS
LIN {X 96.840,Y -17.308,Z -208.172,A -90.000,B 90.000,C 0.000} C_DIS
LIN {X 96.515,Y -17.308,Z -209.595,A -90.000,B 90.000,C 0.000} C_DIS
LIN {X 95.639,Y -17.308,Z -213.568,A -90.000,B 90.000,C 0.000} C_DIS
LIN {X 95.325,Y -17.308,Z -214.886,A -90.000,B 90.000,C 0.000} C_DIS
LIN {X 94.307,Y -17.308,Z -219.216,A -90.000,B 90.000,C 0.000} C_DIS
LIN {X 93.966,Y -17.308,Z -220.619,A -90.000,B 90.000,C 0.000} C_DIS
LIN {X 92.561,Y -17.308,Z -226.171,A -90.000,B 90.000,C 0.000} C_DIS
LIN {X 90.998,Y -17.308,Z -231.834,A -90.000,B 90.000,C 0.000} C_DIS
LIN {X 89.225,Y -17.308,Z -237.703,A -90.000,B 90.000,C 0.000} C_DIS
LIN {X 89.129,Y -17.308,Z -238.013,A -90.000,B 90.000,C 0.000} C_DIS
LIN {X 87.297,Y -17.308,Z -243.561,A -90.000,B 90.000,C 0.000} C_DIS
LIN {X 87.297,Y -60.000,Z -243.561,A -90.000,B 90.000,C 0.000} C_DIS
LIN {X 100.035,Y -60.000,Z -89.825,A -90.000,B 90.000,C 0.000} C_DIS
LIN {X 100.035,Y -15.308,Z -89.825,A -90.000,B 90.000,C 0.000} C_DIS
LIN {X 100.314,Y -15.312,Z -90.386,A -90.000,B 90.000,C 0.000} C_DIS
LIN {X 100.436,Y -15.313,Z -90.693,A -90.000,B 90.000,C 0.000} C_DIS
LIN {X 100.838,Y -15.319,Z -91.630,A -90.000,B 90.000,C 0.000} C_DIS
LIN {X 101.018,Y -15.324,Z -92.110,A -90.000,B 90.000,C 0.000} C_DIS
LIN {X 101.057,Y -15.325,Z -92.218,A -90.000,B 90.000,C 0.000} C_DIS
LIN {X 101.380,Y -15.335,Z -93.201,A -90.000,B 90.000,C 0.000} C_DIS
LIN {X 101.457,Y -15.338,Z -93.475,A -90.000,B 90.000,C 0.000} C_DIS
LIN {X 101.548,Y -15.344,Z -93.813,A -90.000,B 90.000,C 0.000} C_DIS
LIN {X 101.634,Y -15.348,Z -94.137,A -90.000,B 90.000,C 0.000} C_DIS
LIN {X 101.766,Y -15.354,Z -94.670,A -90.000,B 90.000,C 0.000} C_DIS
LIN {X 101.836,Y -15.359,Z -94.969,A -90.000,B 90.000,C 0.000} C_DIS
LIN {X 101.876,Y -15.364,Z -95.146,A -90.000,B 90.000,C 0.000} C_DIS
LIN {X 102.020,Y -15.373,Z -95.895,A -90.000,B 90.000,C 0.000} C_DIS
LIN {X 102.077,Y -15.377,Z -96.171,A -90.000,B 90.000,C 0.000} C_DIS
LIN {X 102.099,Y -15.381,Z -96.310,A -90.000,B 90.000,C 0.000} C_DIS
LIN {X 102.215,Y -15.389,Z -96.991,A -90.000,B 90.000,C 0.000} C_DIS
LIN {X 102.266,Y -15.394,Z -97.241,A -90.000,B 90.000,C 0.000} C_DIS
LIN {X 102.430,Y -15.404,Z -98.165,A -90.000,B 90.000,C 0.000} C_DIS
LIN {X 102.550,Y -15.416,Z -98.762,A -90.000,B 90.000,C 0.000} C_DIS
LIN {X 102.686,Y -15.423,Z -99.523,A -90.000,B 90.000,C 0.000} C_DIS
LIN {X 102.791,Y -15.433,Z -100.078,A -90.000,B 90.000,C 0.000} C_DIS
LIN {X 103.033,Y -15.443,Z -101.449,A -90.000,B 90.000,C 0.000} C_DIS
LIN {X 103.062,Y -15.448,Z -101.621,A -90.000,B 90.000,C 0.000} C_DIS
LIN {X 103.298,Y -15.455,Z -103.020,A -90.000,B 90.000,C 0.000} C_DIS
LIN {X 103.414,Y -15.458,Z -103.738,A -90.000,B 90.000,C 0.000} C_DIS
LIN {X 103.522,Y -15.459,Z -104.415,A -90.000,B 90.000,C 0.000} C_DIS
LIN {X 103.719,Y -15.461,Z -105.621,A -90.000,B 90.000,C 0.000} C_DIS
LIN {X 104.048,Y -15.463,Z -107.776,A -90.000,B 90.000,C 0.000} C_DIS
LIN {X 104.145,Y -15.463,Z -108.429,A -90.000,B 90.000,C 0.000} C_DIS
LIN {X 104.360,Y -15.463,Z -109.974,A -90.000,B 90.000,C 0.000} C_DIS
LIN {X 104.503,Y -15.463,Z -111.018,A -90.000,B 90.000,C 0.000} C_DIS
LIN {X 104.621,Y -15.462,Z -111.962,A -90.000,B 90.000,C 0.000} C_DIS
LIN {X 104.831,Y -15.460,Z -113.677,A -90.000,B 90.000,C 0.000} C_DIS
LIN {X 104.897,Y -15.458,Z -114.294,A -90.000,B 90.000,C 0.000} C_DIS
LIN {X 105.032,Y -15.454,Z -115.592,A -90.000,B 90.000,C 0.000} C_DIS
LIN {X 105.117,Y -15.450,Z -116.411,A -90.000,B 90.000,C 0.000} C_DIS
LIN {X 105.191,Y -15.447,Z -117.233,A -90.000,B 90.000,C 0.000} C_DIS
LIN {X 105.354,Y -15.436,Z -119.050,A -90.000,B 90.000,C 0.000} C_DIS
LIN {X 105.497,Y -15.425,Z -120.836,A -90.000,B 90.000,C 0.000} C_DIS
LIN {X 105.559,Y -15.422,Z -121.547,A -90.000,B 90.000,C 0.000} C_DIS
LIN {X 105.632,Y -15.418,Z -122.593,A -90.000,B 90.000,C 0.000} C_DIS
LIN {X 105.744,Y -15.413,Z -124.082,A -90.000,B 90.000,C 0.000} C_DIS
LIN {X 105.851,Y -15.410,Z -125.788,A -90.000,B 90.000,C 0.000} C_DIS
LIN {X 105.901,Y -15.409,Z -126.610,A -90.000,B 90.000,C 0.000} C_DIS
LIN {X 105.923,Y -15.409,Z -127.030,A -90.000,B 90.000,C 0.000} C_DIS
LIN {X 106.037,Y -15.409,Z -129.551,A -90.000,B 90.000,C 0.000} C_DIS
LIN {X 106.102,Y -15.413,Z -132.223,A -90.000,B 90.000,C 0.000} C_DIS
LIN {X 106.109,Y -15.419,Z -135.132,A -90.000,B 90.000,C 0.000} C_DIS
LIN {X 106.078,Y -15.423,Z -137.064,A -90.000,B 90.000,C 0.000} C_DIS
LIN {X 106.051,Y -15.426,Z -138.497,A -90.000,B 90.000,C 0.000} C_DIS
LIN {X 105.999,Y -15.430,Z -140.171,A -90.000,B 90.000,C 0.000} C_DIS
LIN {X 105.921,Y -15.432,Z -142.375,A -90.000,B 90.000,C 0.000} C_DIS
LIN {X 105.805,Y -15.435,Z -144.780,A -90.000,B 90.000,C 0.000} C_DIS
LIN {X 105.742,Y -15.436,Z -146.069,A -90.000,B 90.000,C 0.000} C_DIS
LIN {X 105.493,Y -15.437,Z -150.016,A -90.000,B 90.000,C 0.000} C_DIS
LIN {X 105.265,Y -15.434,Z -152.923,A -90.000,B 90.000,C 0.000} C_DIS
LIN {X 105.180,Y -15.433,Z -153.968,A -90.000,B 90.000,C 0.000} C_DIS
LIN {X 104.995,Y -15.430,Z -156.042,A -90.000,B 90.000,C 0.000} C_DIS
LIN {X 104.832,Y -15.425,Z -157.786,A -90.000,B 90.000,C 0.000} C_DIS
LIN {X 104.484,Y -15.419,Z -161.317,A -90.000,B 90.000,C 0.000} C_DIS
LIN {X 104.112,Y -15.411,Z -164.879,A -90.000,B 90.000,C 0.000} C_DIS
LIN {X 103.754,Y -15.404,Z -168.227,A -90.000,B 90.000,C 0.000} C_DIS
LIN {X 103.379,Y -15.395,Z -171.600,A -90.000,B 90.000,C 0.000} C_DIS
LIN {X 103.002,Y -15.388,Z -174.799,A -90.000,B 90.000,C 0.000} C_DIS
LIN {X 102.939,Y -15.386,Z -175.305,A -90.000,B 90.000,C 0.000} C_DIS
LIN {X 102.622,Y -15.381,Z -177.777,A -90.000,B 90.000,C 0.000} C_DIS
LIN {X 102.542,Y -15.379,Z -178.373,A -90.000,B 90.000,C 0.000} C_DIS
LIN {X 102.499,Y -15.379,Z -178.673,A -90.000,B 90.000,C 0.000} C_DIS
LIN {X 102.101,Y -15.375,Z -181.454,A -90.000,B 90.000,C 0.000} C_DIS
LIN {X 101.688,Y -15.373,Z -184.145,A -90.000,B 90.000,C 0.000} C_DIS
LIN {X 100.920,Y -15.373,Z -188.985,A -90.000,B 90.000,C 0.000} C_DIS
LIN {X 100.557,Y -15.374,Z -191.391,A -90.000,B 90.000,C 0.000} C_DIS
LIN {X 100.107,Y -15.378,Z -194.292,A -90.000,B 90.000,C 0.000} C_DIS
LIN {X 99.966,Y -15.380,Z -195.176,A -90.000,B 90.000,C 0.000} C_DIS
LIN {X 99.581,Y -15.387,Z -197.485,A -90.000,B 90.000,C 0.000} C_DIS
LIN {X 99.430,Y -15.390,Z -198.378,A -90.000,B 90.000,C 0.000} C_DIS
LIN {X 98.701,Y -15.409,Z -202.411,A -90.000,B 90.000,C 0.000} C_DIS
LIN {X 98.193,Y -15.425,Z -204.996,A -90.000,B 90.000,C 0.000} C_DIS
LIN {X 97.773,Y -15.436,Z -207.170,A -90.000,B 90.000,C 0.000} C_DIS
LIN {X 97.537,Y -15.440,Z -208.332,A -90.000,B 90.000,C 0.000} C_DIS
LIN {X 97.238,Y -15.451,Z -209.758,A -90.000,B 90.000,C 0.000} C_DIS
LIN {X 96.435,Y -15.470,Z -213.612,A -90.000,B 90.000,C 0.000} C_DIS
LIN {X 96.109,Y -15.478,Z -215.072,A -90.000,B 90.000,C 0.000} C_DIS
LIN {X 95.205,Y -15.493,Z -219.060,A -90.000,B 90.000,C 0.000} C_DIS
LIN {X 94.846,Y -15.496,Z -220.577,A -90.000,B 90.000,C 0.000} C_DIS
LIN {X 94.764,Y -15.496,Z -220.916,A -90.000,B 90.000,C 0.000} C_DIS
LIN {X 94.418,Y -15.496,Z -222.281,A -90.000,B 90.000,C 0.000} C_DIS
LIN {X 93.374,Y -15.503,Z -226.457,A -90.000,B 90.000,C 0.000} C_DIS
LIN {X 91.814,Y -15.504,Z -232.119,A -90.000,B 90.000,C 0.000} C_DIS
LIN {X 90.040,Y -15.505,Z -237.997,A -90.000,B 90.000,C 0.000} C_DIS
LIN {X 89.946,Y -15.503,Z -238.283,A -90.000,B 90.000,C 0.000} C_DIS
LIN {X 89.522,Y -15.503,Z -239.569,A -90.000,B 90.000,C 0.000} C_DIS
LIN {X 88.215,Y -15.508,Z -243.561,A -90.000,B 90.000,C 0.000} C_DIS
LIN {X 88.215,Y -60.000,Z -243.561,A -90.000,B 90.000,C 0.000} C_DIS
LIN {X -114.841,Y -60.000,Z -243.561,A -90.000,B 90.000,C 0.000} C_DIS
LIN {X -114.841,Y -16.522,Z -243.561,A -90.000,B 90.000,C 0.000} C_DIS
LIN {X -114.746,Y -16.379,Z -243.257,A -90.000,B 90.000,C 0.000} C_DIS
LIN {X -114.709,Y -16.341,Z -243.176,A -90.000,B 90.000,C 0.000} C_DIS
LIN {X -114.623,Y -16.272,Z -243.015,A -90.000,B 90.000,C 0.000} C_DIS
LIN {X -114.531,Y -16.220,Z -242.872,A -90.000,B 90.000,C 0.000} C_DIS
LIN {X -114.379,Y -16.159,Z -242.677,A -90.000,B 90.000,C 0.000} C_DIS
LIN {X -114.131,Y -16.108,Z -242.429,A -90.000,B 90.000,C 0.000} C_DIS
LIN {X -113.917,Y -16.096,Z -242.261,A -90.000,B 90.000,C 0.000} C_DIS
LIN {X -110.950,Y -16.090,Z -240.177,A -90.000,B 90.000,C 0.000} C_DIS
LIN {X -109.925,Y -16.086,Z -239.454,A -90.000,B 90.000,C 0.000} C_DIS
LIN {X -107.344,Y -16.079,Z -237.627,A -90.000,B 90.000,C 0.000} C_DIS
LIN {X -104.272,Y -16.066,Z -235.472,A -90.000,B 90.000,C 0.000} C_DIS
LIN {X -99.693,Y -16.045,Z -232.266,A -90.000,B 90.000,C 0.000} C_DIS
LIN {X -97.614,Y -16.037,Z -230.827,A -90.000,B 90.000,C 0.000} C_DIS
LIN {X -96.505,Y -16.031,Z -230.063,A -90.000,B 90.000,C 0.000} C_DIS
LIN {X -92.357,Y -16.022,Z -227.225,A -90.000,B 90.000,C 0.000} C_DIS
LIN {X -91.659,Y -16.022,Z -226.749,A -90.000,B 90.000,C 0.000} C_DIS
LIN {X -89.695,Y -16.020,Z -225.428,A -90.000,B 90.000,C 0.000} C_DIS
LIN {X -84.445,Y -16.012,Z -221.905,A -90.000,B 90.000,C 0.000} C_DIS
LIN {X -83.341,Y -16.011,Z -221.168,A -90.000,B 90.000,C 0.000} C_DIS
LIN {X -76.566,Y -15.977,Z -216.760,A -90.000,B 90.000,C 0.000} C_DIS
LIN {X -75.338,Y -15.967,Z -215.966,A -90.000,B 90.000,C 0.000} C_DIS
LIN {X -71.274,Y -15.931,Z -213.355,A -90.000,B 90.000,C 0.000} C_DIS
LIN {X -67.279,Y -15.899,Z -210.795,A -90.000,B 90.000,C 0.000} C_DIS
LIN {X -63.561,Y -15.867,Z -208.398,A -90.000,B 90.000,C 0.000} C_DIS
LIN {X -59.729,Y -15.830,Z -205.931,A -90.000,B 90.000,C 0.000} C_DIS
LIN {X -57.038,Y -15.806,Z -204.164,A -90.000,B 90.000,C 0.000} C_DIS
LIN {X -53.092,Y -15.785,Z -201.603,A -90.000,B 90.000,C 0.000} C_DIS
LIN {X -52.869,Y -15.785,Z -201.456,A -90.000,B 90.000,C 0.000} C_DIS
LIN {X -50.730,Y -15.770,Z -200.008,A -90.000,B 90.000,C 0.000} C_DIS
LIN {X -47.452,Y -15.760,Z -197.805,A -90.000,B 90.000,C 0.000} C_DIS
LIN {X -46.892,Y -15.761,Z -197.416,A -90.000,B 90.000,C 0.000} C_DIS
LIN {X -42.979,Y -15.742,Z -194.676,A -90.000,B 90.000,C 0.000} C_DIS
LIN {X -42.258,Y -15.741,Z -194.154,A -90.000,B 90.000,C 0.000} C_DIS
LIN {X -40.746,Y -15.732,Z -193.050,A -90.000,B 90.000,C 0.000} C_DIS
LIN {X -38.996,Y -15.715,Z -191.783,A -90.000,B 90.000,C 0.000} C_DIS
LIN {X -38.624,Y -15.715,Z -191.506,A -90.000,B 90.000,C 0.000} C_DIS
LIN {X -35.802,Y -15.692,Z -189.387,A -90.000,B 90.000,C 0.000} C_DIS
LIN {X -33.440,Y -15.676,Z -187.581,A -90.000,B 90.000,C 0.000} C_DIS
LIN {X -32.644,Y -15.676,Z -186.976,A -90.000,B 90.000,C 0.000} C_DIS
LIN {X -30.506,Y -15.663,Z -185.284,A -90.000,B 90.000,C 0.000} C_DIS
LIN {X -29.769,Y -15.663,Z -184.704,A -90.000,B 90.000,C 0.000} C_DIS
LIN {X -27.854,Y -15.654,Z -183.107,A -90.000,B 90.000,C 0.000} C_DIS
LIN {X -27.139,Y -15.653,Z -182.513,A -90.000,B 90.000,C 0.000} C_DIS
LIN {X -27.009,Y -15.656,Z -182.400,A -90.000,B 90.000,C 0.000} C_DIS
LIN {X -25.257,Y -15.646,Z -180.836,A -90.000,B 90.000,C 0.000} C_DIS
LIN {X -24.661,Y -15.645,Z -180.305,A -90.000,B 90.000,C 0.000} C_DIS
LIN {X -24.577,Y -15.647,Z -180.226,A -90.000,B 90.000,C 0.000} C_DIS
LIN {X -24.283,Y -15.648,Z -179.942,A -90.000,B 90.000,C 0.000} C_DIS
LIN {X -22.483,Y -15.639,Z -178.195,A -90.000,B 90.000,C 0.000} C_DIS
LIN {X -22.358,Y -15.642,Z -178.065,A -90.000,B 90.000,C 0.000} C_DIS
LIN {X -21.896,Y -15.642,Z -177.573,A -90.000,B 90.000,C 0.000} C_DIS
LIN {X -20.344,Y -15.636,Z -175.915,A -90.000,B 90.000,C 0.000} C_DIS
LIN {X -20.126,Y -15.644,Z -175.663,A -90.000,B 90.000,C 0.000} C_DIS
LIN {X -18.538,Y -15.639,Z -173.770,A -90.000,B 90.000,C 0.000} C_DIS
LIN {X -18.321,Y -15.648,Z -173.486,A -90.000,B 90.000,C 0.000} C_DIS
LIN {X -17.965,Y -15.649,Z -173.007,A -90.000,B 90.000,C 0.000} C_DIS
LIN {X -16.777,Y -15.643,Z -171.395,A -90.000,B 90.000,C 0.000} C_DIS
LIN {X -16.529,Y -15.655,Z -171.025,A -90.000,B 90.000,C 0.000} C_DIS
LIN {X -15.232,Y -15.642,Z -168.990,A -90.000,B 90.000,C 0.000} C_DIS
LIN {X -15.075,Y -15.654,Z -168.704,A -90.000,B 90.000,C 0.000} C_DIS
LIN {X -14.969,Y -15.662,Z -168.516,A -90.000,B 90.000,C 0.000} C_DIS
LIN {X -13.965,Y -15.644,Z -166.630,A -90.000,B 90.000,C 0.000} C_DIS
LIN {X -13.778,Y -15.668,Z -166.196,A -90.000,B 90.000,C 0.000} C_DIS
LIN {X -13.713,Y -15.668,Z -166.029,A -90.000,B 90.000,C 0.000} C_DIS
LIN {X -13.092,Y -15.651,Z -164.518,A -90.000,B 90.000,C 0.000} C_DIS
LIN {X -13.006,Y -15.674,Z -164.206,A -90.000,B 90.000,C 0.000} C_DIS
LIN {X -12.953,Y -15.672,Z -163.992,A -90.000,B 90.000,C 0.000} C_DIS
LIN {X -12.698,Y -15.651,Z -162.968,A -90.000,B 90.000,C 0.000} C_DIS
LIN {X -12.687,Y -15.664,Z -162.828,A -90.000,B 90.000,C 0.000} C_DIS
LIN {X -12.682,Y -15.643,Z -162.100,A -90.000,B 90.000,C 0.000} C_DIS
LIN {X -12.685,Y -15.636,Z -162.057,A -90.000,B 90.000,C 0.000} C_DIS
LIN {X -12.707,Y -15.635,Z -161.980,A -90.000,B 90.000,C 0.000} C_DIS
LIN {X -12.773,Y -15.626,Z -161.732,A -90.000,B 90.000,C 0.000} C_DIS
LIN {X -12.862,Y -15.588,Z -161.467,A -90.000,B 90.000,C 0.000} C_DIS
LIN {X -12.870,Y -15.587,Z -161.452,A -90.000,B 90.000,C 0.000} C_DIS
LIN {X -13.049,Y -15.575,Z -161.113,A -90.000,B 90.000,C 0.000} C_DIS
LIN {X -13.247,Y -15.539,Z -160.769,A -90.000,B 90.000,C 0.000} C_DIS
LIN {X -13.336,Y -15.534,Z -160.644,A -90.000,B 90.000,C 0.000} C_DIS
LIN {X -13.588,Y -15.527,Z -160.287,A -90.000,B 90.000,C 0.000} C_DIS
LIN {X -13.726,Y -15.525,Z -160.088,A -90.000,B 90.000,C 0.000} C_DIS
LIN {X -13.903,Y -15.511,Z -159.845,A -90.000,B 90.000,C 0.000} C_DIS
LIN {X -14.037,Y -15.505,Z -159.675,A -90.000,B 90.000,C 0.000} C_DIS
LIN {X -14.255,Y -15.494,Z -159.391,A -90.000,B 90.000,C 0.000} C_DIS
LIN {X -14.595,Y -15.490,Z -158.937,A -90.000,B 90.000,C 0.000} C_DIS
LIN {X -14.777,Y -15.476,Z -158.702,A -90.000,B 90.000,C 0.000} C_DIS
LIN {X -15.267,Y -15.456,Z -158.122,A -90.000,B 90.000,C 0.000} C_DIS
LIN {X -15.658,Y -15.455,Z -157.653,A -90.000,B 90.000,C 0.000} C_DIS
LIN {X -15.773,Y -15.447,Z -157.514,A -90.000,B 90.000,C 0.000} C_DIS
LIN {X -16.269,Y -15.435,Z -156.989,A -90.000,B 90.000,C 0.000} C_DIS
LIN {X -16.724,Y -15.431,Z -156.504,A -90.000,B 90.000,C 0.000} C_DIS
LIN {X -17.090,Y -15.430,Z -156.112,A -90.000,B 90.000,C 0.000} C_DIS
LIN {X -17.166,Y -15.428,Z -156.032,A -90.000,B 90.000,C 0.000} C_DIS
LIN {X -17.277,Y -15.424,Z -155.913,A -90.000,B 90.000,C 0.000} C_DIS
LIN {X -18.273,Y -15.409,Z -154.943,A -90.000,B 90.000,C 0.000} C_DIS
LIN {X -19.046,Y -15.409,Z -154.186,A -90.000,B 90.000,C 0.000} C_DIS
LIN {X -19.173,Y -15.406,Z -154.062,A -90.000,B 90.000,C 0.000} C_DIS
LIN {X -20.735,Y -15.393,Z -152.632,A -90.000,B 90.000,C 0.000} C_DIS
LIN {X -21.607,Y -15.392,Z -151.832,A -90.000,B 90.000,C 0.000} C_DIS
LIN {X -21.935,Y -15.391,Z -151.524,A -90.000,B 90.000,C 0.000} C_DIS
LIN {X -23.747,Y -15.381,Z -149.813,A -90.000,B 90.000,C 0.000} C_DIS
LIN {X -25.057,Y -15.381,Z -148.573,A -90.000,B 90.000,C 0.000} C_DIS
LIN {X -25.245,Y -15.381,Z -148.391,A -90.000,B 90.000,C 0.000} C_DIS
LIN {X -25.778,Y -15.378,Z -147.839,A -90.000,B 90.000,C 0.000} C_DIS
LIN {X -27.403,Y -15.372,Z -146.151,A -90.000,B 90.000,C 0.000} C_DIS
LIN {X -28.528,Y -15.371,Z -144.978,A -90.000,B 90.000,C 0.000} C_DIS
LIN {X -28.785,Y -15.371,Z -144.696,A -90.000,B 90.000,C 0.000} C_DIS
LIN {X -29.051,Y -15.370,Z -144.377,A -90.000,B 90.000,C 0.000} C_DIS
LIN {X -31.833,Y -15.362,Z -140.980,A -90.000,B 90.000,C 0.000} C_DIS
LIN {X -32.109,Y -15.361,Z -140.608,A -90.000,B 90.000,C 0.000} C_DIS
LIN {X -32.175,Y -15.360,Z -140.507,A -90.000,B 90.000,C 0.000} C_DIS
LIN {X -34.103,Y -15.355,Z -137.461,A -90.000,B 90.000,C 0.000} C_DIS
LIN {X -34.650,Y -15.355,Z -136.610,A -90.000,B 90.000,C 0.000} C_DIS
LIN {X -34.896,Y -15.354,Z -136.195,A -90.000,B 90.000,C 0.000} C_DIS
LIN {X -36.249,Y -15.355,Z -133.577,A -90.000,B 90.000,C 0.000} C_DIS
LIN {X -36.954,Y -15.357,Z -132.225,A -90.000,B 90.000,C 0.000} C_DIS
LIN {X -37.031,Y -15.356,Z -132.058,A -90.000,B 90.000,C 0.000} C_DIS
LIN {X -37.156,Y -15.355,Z -131.787,A -90.000,B 90.000,C 0.000} C_DIS
LIN {X -37.982,Y -15.358,Z -129.922,A -90.000,B 90.000,C 0.000} C_DIS
LIN {X -38.793,Y -15.363,Z -128.103,A -90.000,B 90.000,C 0.000} C_DIS
LIN {X -39.216,Y -15.362,Z -127.054,A -90.000,B 90.000,C 0.000} C_DIS
LIN {X -39.925,Y -15.363,Z -125.310,A -90.000,B 90.000,C 0.000} C_DIS
LIN {X -40.215,Y -15.365,Z -124.601,A -90.000,B 90.000,C 0.000} C_DIS
LIN {X -41.013,Y -15.359,Z -122.667,A -90.000,B 90.000,C 0.000} C_DIS
LIN {X -41.088,Y -15.358,Z -122.503,A -90.000,B 90.000,C 0.000} C_DIS
LIN {X -41.516,Y -15.353,Z -121.571,A -90.000,B 90.000,C 0.000} C_DIS
LIN {X -41.689,Y -15.350,Z -121.219,A -90.000,B 90.000,C 0.000} C_DIS
LIN {X -41.753,Y -15.351,Z -121.106,A -90.000,B 90.000,C 0.000} C_DIS
LIN {X -42.200,Y -15.345,Z -120.331,A -90.000,B 90.000,C 0.000} C_DIS
LIN {X -42.430,Y -15.343,Z -119.954,A -90.000,B 90.000,C 0.000} C_DIS
LIN {X -42.527,Y -15.345,Z -119.818,A -90.000,B 90.000,C 0.000} C_DIS
LIN {X -43.062,Y -15.342,Z -119.063,A -90.000,B 90.000,C 0.000} C_DIS
LIN {X -43.494,Y -15.340,Z -118.473,A -90.000,B 90.000,C 0.000} C_DIS
LIN {X -44.842,Y -15.342,Z -116.805,A -90.000,B 90.000,C 0.000} C_DIS
LIN {X -45.302,Y -15.341,Z -116.233,A -90.000,B 90.000,C 0.000} C_DIS
LIN {X -47.537,Y -15.348,Z -113.547,A -90.000,B 90.000,C 0.000} C_DIS
LIN {X -50.011,Y -15.356,Z -110.523,A -90.000,B 90.000,C 0.000} C_DIS
LIN {X -50.348,Y -15.355,Z -110.094,A -90.000,B 90.000,C 0.000} C_DIS
LIN {X -51.130,Y -15.357,Z -109.097,A -90.000,B 90.000,C 0.000} C_DIS
LIN {X -52.563,Y -15.362,Z -107.277,A -90.000,B 90.000,C 0.000} C_DIS
LIN {X -52.959,Y -15.360,Z -106.743,A -90.000,B 90.000,C 0.000} C_DIS
LIN {X -55.057,Y -15.363,Z -103.901,A -90.000,B 90.000,C 0.000} C_DIS
LIN {X -55.365,Y -15.363,Z -103.480,A -90.000,B 90.000,C 0.000} C_DIS
LIN {X -56.910,Y -15.358,Z -101.320,A -90.000,B 90.000,C 0.000} C_DIS
LIN {X -58.529,Y -15.355,Z -99.079,A -90.000,B 90.000,C 0.000} C_DIS
LIN {X -58.694,Y -15.355,Z -98.853,A -90.000,B 90.000,C 0.000} C_DIS
LIN {X -59.889,Y -15.351,Z -97.212,A -90.000,B 90.000,C 0.000} C_DIS
LIN {X -59.995,Y -15.351,Z -97.071,A -90.000,B 90.000,C 0.000} C_DIS
LIN {X -61.929,Y -15.347,Z -94.516,A -90.000,B 90.000,C 0.000} C_DIS
LIN {X -62.142,Y -15.349,Z -94.255,A -90.000,B 90.000,C 0.000} C_DIS
LIN {X -62.795,Y -15.352,Z -93.457,A -90.000,B 90.000,C 0.000} C_DIS
LIN {X -63.877,Y -15.351,Z -92.109,A -90.000,B 90.000,C 0.000} C_DIS
LIN {X -64.340,Y -15.359,Z -91.594,A -90.000,B 90.000,C 0.000} C_DIS
LIN {X -64.721,Y -15.361,Z -91.171,A -90.000,B 90.000,C 0.000} C_DIS
LIN {X -65.596,Y -15.362,Z -90.164,A -90.000,B 90.000,C 0.000} C_DIS
LIN {X -66.112,Y -15.376,Z -89.647,A -90.000,B 90.000,C 0.000} C_DIS
LIN {X -66.254,Y -15.378,Z -89.505,A -90.000,B 90.000,C 0.000} C_DIS
LIN {X -67.262,Y -15.385,Z -88.450,A -90.000,B 90.000,C 0.000} C_DIS
LIN {X -67.778,Y -15.405,Z -87.986,A -90.000,B 90.000,C 0.000} C_DIS
LIN {X -68.152,Y -15.411,Z -87.654,A -90.000,B 90.000,C 0.000} C_DIS
LIN {X -68.413,Y -15.413,Z -87.408,A -90.000,B 90.000,C 0.000} C_DIS
LIN {X -69.091,Y -15.424,Z -86.769,A -90.000,B 90.000,C 0.000} C_DIS
LIN {X -69.497,Y -15.441,Z -86.422,A -90.000,B 90.000,C 0.000} C_DIS
LIN {X -70.208,Y -15.459,Z -85.820,A -90.000,B 90.000,C 0.000} C_DIS
LIN {X -70.820,Y -15.480,Z -85.316,A -90.000,B 90.000,C 0.000} C_DIS
LIN {X -71.069,Y -15.492,Z -85.120,A -90.000,B 90.000,C 0.000} C_DIS
LIN {X -72.134,Y -15.528,Z -84.288,A -90.000,B 90.000,C 0.000} C_DIS
LIN {X -72.761,Y -15.554,Z -83.811,A -90.000,B 90.000,C 0.000} C_DIS
LIN {X -72.952,Y -15.560,Z -83.668,A -90.000,B 90.000,C 0.000} C_DIS
LIN {X -73.092,Y -15.565,Z -83.567,A -90.000,B 90.000,C 0.000} C_DIS
LIN {X -74.304,Y -15.603,Z -82.703,A -90.000,B 90.000,C 0.000} C_DIS
LIN {X -74.379,Y -15.604,Z -82.651,A -90.000,B 90.000,C 0.000} C_DIS
LIN {X -74.705,Y -15.611,Z -82.424,A -90.000,B 90.000,C 0.000} C_DIS
LIN {X -74.889,Y -15.619,Z -82.305,A -90.000,B 90.000,C 0.000} C_DIS
LIN {X -75.284,Y -15.625,Z -82.058,A -90.000,B 90.000,C 0.000} C_DIS
LIN {X -76.473,Y -15.629,Z -81.325,A -90.000,B 90.000,C 0.000} C_DIS
LIN {X -76.740,Y -15.616,Z -81.171,A -90.000,B 90.000,C 0.000} C_DIS
LIN {X -77.359,Y -15.599,Z -80.842,A -90.000,B 90.000,C 0.000} C_DIS
LIN {X -77.832,Y -15.587,Z -80.598,A -90.000,B 90.000,C 0.000} C_DIS
LIN {X -78.328,Y -15.565,Z -80.350,A -90.000,B 90.000,C 0.000} C_DIS
LIN {X -79.408,Y -15.527,Z -79.808,A -90.000,B 90.000,C 0.000} C_DIS
LIN {X -79.711,Y -15.514,Z -79.657,A -90.000,B 90.000,C 0.000} C_DIS
LIN {X -79.937,Y -15.510,Z -79.547,A -90.000,B 90.000,C 0.000} C_DIS
LIN {X -80.330,Y -15.500,Z -79.345,A -90.000,B 90.000,C 0.000} C_DIS
LIN {X -81.282,Y -15.471,Z -78.843,A -90.000,B 90.000,C 0.000} C_DIS
LIN {X -81.691,Y -15.468,Z -78.621,A -90.000,B 90.000,C 0.000} C_DIS
LIN {X -81.912,Y -15.470,Z -78.504,A -90.000,B 90.000,C 0.000} C_DIS
LIN {X -82.161,Y -15.465,Z -78.353,A -90.000,B 90.000,C 0.000} C_DIS
LIN {X -83.187,Y -15.432,Z -77.724,A -90.000,B 90.000,C 0.000} C_DIS
LIN {X -83.437,Y -15.428,Z -77.560,A -90.000,B 90.000,C 0.000} C_DIS
LIN {X -83.619,Y -15.427,Z -77.445,A -90.000,B 90.000,C 0.000} C_DIS
LIN {X -83.814,Y -15.422,Z -77.305,A -90.000,B 90.000,C 0.000} C_DIS
LIN {X -83.918,Y -15.418,Z -77.228,A -90.000,B 90.000,C 0.000} C_DIS
LIN {X -84.266,Y -15.408,Z -76.971,A -90.000,B 90.000,C 0.000} C_DIS
LIN {X -84.752,Y -15.403,Z -76.608,A -90.000,B 90.000,C 0.000} C_DIS
LIN {X -85.208,Y -15.394,Z -76.248,A -90.000,B 90.000,C 0.000} C_DIS
LIN {X -85.535,Y -15.386,Z -75.982,A -90.000,B 90.000,C 0.000} C_DIS
LIN {X -86.255,Y -15.377,Z -75.388,A -90.000,B 90.000,C 0.000} C_DIS
LIN {X -86.940,Y -15.366,Z -74.813,A -90.000,B 90.000,C 0.000} C_DIS
LIN {X -87.298,Y -15.363,Z -74.514,A -90.000,B 90.000,C 0.000} C_DIS
LIN {X -87.603,Y -15.359,Z -74.263,A -90.000,B 90.000,C 0.000} C_DIS
LIN {X -87.904,Y -15.360,Z -74.037,A -90.000,B 90.000,C 0.000} C_DIS
LIN {X -88.351,Y -15.360,Z -73.687,A -90.000,B 90.000,C 0.000} C_DIS
LIN {X -88.716,Y -15.369,Z -73.438,A -90.000,B 90.000,C 0.000} C_DIS
LIN {X -89.001,Y -15.374,Z -73.228,A -90.000,B 90.000,C 0.000} C_DIS
LIN {X -89.540,Y -15.400,Z -72.891,A -90.000,B 90.000,C 0.000} C_DIS
LIN {X -89.618,Y -15.404,Z -72.839,A -90.000,B 90.000,C 0.000} C_DIS
LIN {X -90.077,Y -15.437,Z -72.575,A -90.000,B 90.000,C 0.000} C_DIS
LIN {X -90.391,Y -15.469,Z -72.424,A -90.000,B 90.000,C 0.000} C_DIS
LIN {X -90.865,Y -15.518,Z -72.175,A -90.000,B 90.000,C 0.000} C_DIS
LIN {X -90.892,Y -15.521,Z -72.162,A -90.000,B 90.000,C 0.000} C_DIS
LIN {X -91.053,Y -15.539,Z -72.088,A -90.000,B 90.000,C 0.000} C_DIS
LIN {X -91.458,Y -15.586,Z -71.901,A -90.000,B 90.000,C 0.000} C_DIS
LIN {X -91.571,Y -15.595,Z -71.850,A -90.000,B 90.000,C 0.000} C_DIS
LIN {X -91.794,Y -15.616,Z -71.755,A -90.000,B 90.000,C 0.000} C_DIS
LIN {X -92.050,Y -15.635,Z -71.651,A -90.000,B 90.000,C 0.000} C_DIS
LIN {X -92.465,Y -15.667,Z -71.479,A -90.000,B 90.000,C 0.000} C_DIS
LIN {X -92.655,Y -15.678,Z -71.404,A -90.000,B 90.000,C 0.000} C_DIS
LIN {X -93.337,Y -15.719,Z -71.127,A -90.000,B 90.000,C 0.000} C_DIS
LIN {X -93.458,Y -15.728,Z -71.075,A -90.000,B 90.000,C 0.000} C_DIS
LIN {X -93.514,Y -15.735,Z -71.054,A -90.000,B 90.000,C 0.000} C_DIS
LIN {X -93.787,Y -15.759,Z -70.954,A -90.000,B 90.000,C 0.000} C_DIS
LIN {X -93.921,Y -15.772,Z -70.906,A -90.000,B 90.000,C 0.000} C_DIS
LIN {X -94.121,Y -15.790,Z -70.831,A -90.000,B 90.000,C 0.000} C_DIS
LIN {X -94.488,Y -15.831,Z -70.688,A -90.000,B 90.000,C 0.000} C_DIS
LIN {X -94.656,Y -15.853,Z -70.620,A -90.000,B 90.000,C 0.000} C_DIS
LIN {X -94.899,Y -15.870,Z -70.532,A -90.000,B 90.000,C 0.000} C_DIS
LIN {X -95.144,Y -15.885,Z -70.438,A -90.000,B 90.000,C 0.000} C_DIS
LIN {X -95.324,Y -15.903,Z -70.361,A -90.000,B 90.000,C 0.000} C_DIS
LIN {X -95.429,Y -15.918,Z -70.326,A -90.000,B 90.000,C 0.000} C_DIS
LIN {X -95.462,Y -15.922,Z -70.313,A -90.000,B 90.000,C 0.000} C_DIS
LIN {X -95.514,Y -15.923,Z -70.297,A -90.000,B 90.000,C 0.000} C_DIS
LIN {X -95.680,Y -15.931,Z -70.241,A -90.000,B 90.000,C 0.000} C_DIS
LIN {X -95.841,Y -15.944,Z -70.180,A -90.000,B 90.000,C 0.000} C_DIS
LIN {X -96.468,Y -16.000,Z -69.994,A -90.000,B 90.000,C 0.000} C_DIS
LIN {X -96.576,Y -16.005,Z -69.957,A -90.000,B 90.000,C 0.000} C_DIS
LIN {X -96.927,Y -16.026,Z -69.823,A -90.000,B 90.000,C 0.000} C_DIS
LIN {X -97.028,Y -16.023,Z -69.794,A -90.000,B 90.000,C 0.000} C_DIS
LIN {X -97.397,Y -16.023,Z -69.676,A -90.000,B 90.000,C 0.000} C_DIS
LIN {X -98.002,Y -16.035,Z -69.470,A -90.000,B 90.000,C 0.000} C_DIS
LIN {X -98.401,Y -16.020,Z -69.314,A -90.000,B 90.000,C 0.000} C_DIS
LIN {X -98.634,Y -16.016,Z -69.217,A -90.000,B 90.000,C 0.000} C_DIS
LIN {X -98.922,Y -16.019,Z -69.089,A -90.000,B 90.000,C 0.000} C_DIS
LIN {X -99.548,Y -16.036,Z -68.798,A -90.000,B 90.000,C 0.000} C_DIS
LIN {X -100.199,Y -16.014,Z -68.447,A -90.000,B 90.000,C 0.000} C_DIS
LIN {X -100.532,Y -16.017,Z -68.250,A -90.000,B 90.000,C 0.000} C_DIS
LIN {X -100.581,Y -16.021,Z -68.222,A -90.000,B 90.000,C 0.000} C_DIS
LIN {X -100.683,Y -16.022,Z -68.160,A -90.000,B 90.000,C 0.000} C_DIS
LIN {X -101.076,Y -16.038,Z -67.911,A -90.000,B 90.000,C 0.000} C_DIS
LIN {X -101.331,Y -16.030,Z -67.731,A -90.000,B 90.000,C 0.000} C_DIS
LIN {X -101.751,Y -16.013,Z -67.429,A -90.000,B 90.000,C 0.000} C_DIS
LIN {X -101.866,Y -16.012,Z -67.342,A -90.000,B 90.000,C 0.000} C_DIS
LIN {X -102.240,Y -16.019,Z -67.042,A -90.000,B 90.000,C 0.000} C_DIS
LIN {X -102.316,Y -16.022,Z -66.980,A -90.000,B 90.000,C 0.000} C_DIS
LIN {X -102.568,Y -16.035,Z -66.764,A -90.000,B 90.000,C 0.000} C_DIS
LIN {X -102.769,Y -16.033,Z -66.577,A -90.000,B 90.000,C 0.000} C_DIS
LIN {X -103.295,Y -16.012,Z -66.053,A -90.000,B 90.000,C 0.000} C_DIS
LIN {X -103.458,Y -16.010,Z -65.883,A -90.000,B 90.000,C 0.000} C_DIS
LIN {X -103.618,Y -16.011,Z -65.712,A -90.000,B 90.000,C 0.000} C_DIS
LIN {X -103.723,Y -16.017,Z -65.594,A -90.000,B 90.000,C 0.000} C_DIS
LIN {X -103.842,Y -16.025,Z -65.448,A -90.000,B 90.000,C 0.000} C_DIS
LIN {X -103.962,Y -16.033,Z -65.293,A -90.000,B 90.000,C 0.000} C_DIS
LIN {X -104.125,Y -16.036,Z -65.072,A -90.000,B 90.000,C 0.000} C_DIS
LIN {X -104.281,Y -16.037,Z -64.857,A -90.000,B 90.000,C 0.000} C_DIS
LIN {X -104.659,Y -16.036,Z -64.328,A -90.000,B 90.000,C 0.000} C_DIS
LIN {X -104.853,Y -16.040,Z -64.048,A -90.000,B 90.000,C 0.000} C_DIS
LIN {X -105.210,Y -16.040,Z -63.523,A -90.000,B 90.000,C 0.000} C_DIS
LIN {X -105.273,Y -16.043,Z -63.425,A -90.000,B 90.000,C 0.000} C_DIS
LIN {X -105.367,Y -16.050,Z -63.274,A -90.000,B 90.000,C 0.000} C_DIS
LIN {X -105.455,Y -16.054,Z -63.122,A -90.000,B 90.000,C 0.000} C_DIS
LIN {X -105.612,Y -16.062,Z -62.842,A -90.000,B 90.000,C 0.000} C_DIS
LIN {X -105.791,Y -16.071,Z -62.508,A -90.000,B 90.000,C 0.000} C_DIS
LIN {X -105.981,Y -16.069,Z -62.126,A -90.000,B 90.000,C 0.000} C_DIS
LIN {X -106.241,Y -16.067,Z -61.599,A -90.000,B 90.000,C 0.000} C_DIS
LIN {X -106.433,Y -16.061,Z -61.196,A -90.000,B 90.000,C 0.000} C_DIS
LIN {X -106.490,Y -16.060,Z -61.071,A -90.000,B 90.000,C 0.000} C_DIS
LIN {X -106.559,Y -16.061,Z -60.907,A -90.000,B 90.000,C 0.000} C_DIS
LIN {X -106.736,Y -16.053,Z -60.505,A -90.000,B 90.000,C 0.000} C_DIS
LIN {X -106.754,Y -16.048,Z -60.476,A -90.000,B 90.000,C 0.000} C_DIS
LIN {X -106.933,Y -15.994,Z -60.196,A -90.000,B 90.000,C 0.000} C_DIS
LIN {X -107.071,Y -15.951,Z -59.974,A -90.000,B 90.000,C 0.000} C_DIS
LIN {X -107.309,Y -15.879,Z -59.577,A -90.000,B 90.000,C 0.000} C_DIS
LIN {X -107.425,Y -15.840,Z -59.376,A -90.000,B 90.000,C 0.000} C_DIS
LIN {X -107.632,Y -15.767,Z -58.998,A -90.000,B 90.000,C 0.000} C_DIS
LIN {X -107.696,Y -15.746,Z -58.877,A -90.000,B 90.000,C 0.000} C_DIS
LIN {X -108.014,Y -15.634,Z -58.244,A -90.000,B 90.000,C 0.000} C_DIS
LIN {X -108.147,Y -15.588,Z -57.960,A -90.000,B 90.000,C 0.000} C_DIS
LIN {X -108.225,Y -15.561,Z -57.781,A -90.000,B 90.000,C 0.000} C_DIS
LIN {X -108.342,Y -15.518,Z -57.498,A -90.000,B 90.000,C 0.000} C_DIS
LIN {X -108.455,Y -15.483,Z -57.219,A -90.000,B 90.000,C 0.000} C_DIS
LIN {X -108.593,Y -15.443,Z -56.876,A -90.000,B 90.000,C 0.000} C_DIS
LIN {X -108.619,Y -15.435,Z -56.804,A -90.000,B 90.000,C 0.000} C_DIS
LIN {X -108.627,Y -15.434,Z -56.790,A -90.000,B 90.000,C 0.000} C_DIS
LIN {X -108.662,Y -15.433,Z -56.734,A -90.000,B 90.000,C 0.000} C_DIS
LIN {X -108.803,Y -15.434,Z -56.542,A -90.000,B 90.000,C 0.000} C_DIS
LIN {X -109.177,Y -15.448,Z -56.041,A -90.000,B 90.000,C 0.000} C_DIS
LIN {X -109.377,Y -15.459,Z -55.767,A -90.000,B 90.000,C 0.000} C_DIS
LIN {X -109.608,Y -15.479,Z -55.466,A -90.000,B 90.000,C 0.000} C_DIS
LIN {X -109.801,Y -15.488,Z -55.183,A -90.000,B 90.000,C 0.000} C_DIS
LIN {X -109.972,Y -15.499,Z -54.941,A -90.000,B 90.000,C 0.000} C_DIS
LIN {X -110.300,Y -15.527,Z -54.453,A -90.000,B 90.000,C 0.000} C_DIS
LIN {X -110.451,Y -15.544,Z -54.214,A -90.000,B 90.000,C 0.000} C_DIS
LIN {X -110.653,Y -15.566,Z -53.868,A -90.000,B 90.000,C 0.000} C_DIS
LIN {X -110.764,Y -15.578,Z -53.660,A -90.000,B 90.000,C 0.000} C_DIS
LIN {X -110.857,Y -15.587,Z -53.491,A -90.000,B 90.000,C 0.000} C_DIS
LIN {X -110.924,Y -15.591,Z -53.357,A -90.000,B 90.000,C 0.000} C_DIS
LIN {X -110.992,Y -15.598,Z -53.215,A -90.000,B 90.000,C 0.000} C_DIS
LIN {X -111.177,Y -15.627,Z -52.798,A -90.000,B 90.000,C 0.000} C_DIS
LIN {X -111.280,Y -15.641,Z -52.552,A -90.000,B 90.000,C 0.000} C_DIS
LIN {X -111.307,Y -15.644,Z -52.484,A -90.000,B 90.000,C 0.000} C_DIS
LIN {X -111.357,Y -15.652,Z -52.350,A -90.000,B 90.000,C 0.000} C_DIS
LIN {X -111.482,Y -15.673,Z -51.930,A -90.000,B 90.000,C 0.000} C_DIS
LIN {X -111.514,Y -15.682,Z -51.794,A -90.000,B 90.000,C 0.000} C_DIS
LIN {X -111.552,Y -15.696,Z -51.629,A -90.000,B 90.000,C 0.000} C_DIS
LIN {X -111.564,Y -15.700,Z -51.561,A -90.000,B 90.000,C 0.000} C_DIS
LIN {X -111.643,Y -15.727,Z -51.093,A -90.000,B 90.000,C 0.000} C_DIS
LIN {X -111.688,Y -15.741,Z -50.788,A -90.000,B 90.000,C 0.000} C_DIS
LIN {X -111.709,Y -15.755,Z -50.621,A -90.000,B 90.000,C 0.000} C_DIS
LIN {X -111.731,Y -15.777,Z -50.201,A -90.000,B 90.000,C 0.000} C_DIS
LIN {X -111.731,Y -15.778,Z -50.157,A -90.000,B 90.000,C 0.000} C_DIS
LIN {X -111.727,Y -15.783,Z -50.054,A -90.000,B 90.000,C 0.000} C_DIS
LIN {X -111.713,Y -15.796,Z -49.803,A -90.000,B 90.000,C 0.000} C_DIS
LIN {X -111.704,Y -15.803,Z -49.669,A -90.000,B 90.000,C 0.000} C_DIS
LIN {X -111.691,Y -15.811,Z -49.529,A -90.000,B 90.000,C 0.000} C_DIS
LIN {X -111.671,Y -15.813,Z -49.391,A -90.000,B 90.000,C 0.000} C_DIS
LIN {X -111.630,Y -15.821,Z -49.131,A -90.000,B 90.000,C 0.000} C_DIS
LIN {X -111.602,Y -15.826,Z -48.967,A -90.000,B 90.000,C 0.000} C_DIS
LIN {X -111.548,Y -15.844,Z -48.677,A -90.000,B 90.000,C 0.000} C_DIS
LIN {X -111.509,Y -15.844,Z -48.527,A -90.000,B 90.000,C 0.000} C_DIS
LIN {X -111.469,Y -15.846,Z -48.374,A -90.000,B 90.000,C 0.000} C_DIS
LIN {X -111.438,Y -15.851,Z -48.272,A -90.000,B 90.000,C 0.000} C_DIS
LIN {X -111.350,Y -15.853,Z -48.024,A -90.000,B 90.000,C 0.000} C_DIS
LIN {X -111.287,Y -15.857,Z -47.846,A -90.000,B 90.000,C 0.000} C_DIS
LIN {X -111.145,Y -15.859,Z -47.479,A -90.000,B 90.000,C 0.000} C_DIS
LIN {X -111.115,Y -15.858,Z -47.413,A -90.000,B 90.000,C 0.000} C_DIS
LIN {X -110.987,Y -15.861,Z -47.150,A -90.000,B 90.000,C 0.000} C_DIS
LIN {X -110.988,Y -15.816,Z -47.053,A -90.000,B 90.000,C 0.000} C_DIS
LIN {X -110.985,Y -15.766,Z -46.935,A -90.000,B 90.000,C 0.000} C_DIS
LIN {X -110.973,Y -15.694,Z -46.758,A -90.000,B 90.000,C 0.000} C_DIS
LIN {X -110.941,Y -15.585,Z -46.458,A -90.000,B 90.000,C 0.000} C_DIS
LIN {X -110.920,Y -15.545,Z -46.343,A -90.000,B 90.000,C 0.000} C_DIS
LIN {X -110.902,Y -15.515,Z -46.252,A -90.000,B 90.000,C 0.000} C_DIS
LIN {X -111.119,Y -15.531,Z -45.847,A -90.000,B 90.000,C 0.000} C_DIS
LIN {X -111.306,Y -15.540,Z -45.477,A -90.000,B 90.000,C 0.000} C_DIS
LIN {X -111.454,Y -15.553,Z -45.172,A -90.000,B 90.000,C 0.000} C_DIS
LIN {X -111.626,Y -15.569,Z -44.790,A -90.000,B 90.000,C 0.000} C_DIS
LIN {X -111.766,Y -15.583,Z -44.447,A -90.000,B 90.000,C 0.000} C_DIS
LIN {X -111.960,Y -15.603,Z -43.963,A -90.000,B 90.000,C 0.000} C_DIS
LIN {X -112.022,Y -15.611,Z -43.804,A -90.000,B 90.000,C 0.000} C_DIS
LIN {X -112.166,Y -15.633,Z -43.369,A -90.000,B 90.000,C 0.000} C_DIS
LIN {X -112.275,Y -15.651,Z -43.007,A -90.000,B 90.000,C 0.000} C_DIS
LIN {X -112.335,Y -15.661,Z -42.788,A -90.000,B 90.000,C 0.000} C_DIS
LIN {X -112.423,Y -15.685,Z -42.441,A -90.000,B 90.000,C 0.000} C_DIS
LIN {X -112.488,Y -15.699,Z -42.109,A -90.000,B 90.000,C 0.000} C_DIS
LIN {X -112.557,Y -15.719,Z -41.715,A -90.000,B 90.000,C 0.000} C_DIS
LIN {X -112.620,Y -15.750,Z -41.305,A -90.000,B 90.000,C 0.000} C_DIS
LIN {X -112.647,Y -15.775,Z -40.955,A -90.000,B 90.000,C 0.000} C_DIS
LIN {X -112.664,Y -15.793,Z -40.608,A -90.000,B 90.000,C 0.000} C_DIS
LIN {X -112.675,Y -15.815,Z -40.252,A -90.000,B 90.000,C 0.000} C_DIS
LIN {X -112.672,Y -15.837,Z -39.959,A -90.000,B 90.000,C 0.000} C_DIS
LIN {X -112.663,Y -15.847,Z -39.764,A -90.000,B 90.000,C 0.000} C_DIS
LIN {X -112.646,Y -15.863,Z -39.528,A -90.000,B 90.000,C 0.000} C_DIS
LIN {X -112.630,Y -15.873,Z -39.346,A -90.000,B 90.000,C 0.000} C_DIS
LIN {X -112.615,Y -15.883,Z -39.231,A -90.000,B 90.000,C 0.000} C_DIS
LIN {X -112.555,Y -15.900,Z -38.895,A -90.000,B 90.000,C 0.000} C_DIS
LIN {X -112.482,Y -15.922,Z -38.517,A -90.000,B 90.000,C 0.000} C_DIS
LIN {X -112.352,Y -15.943,Z -38.064,A -90.000,B 90.000,C 0.000} C_DIS
LIN {X -112.263,Y -15.957,Z -37.774,A -90.000,B 90.000,C 0.000} C_DIS
LIN {X -112.169,Y -15.968,Z -37.515,A -90.000,B 90.000,C 0.000} C_DIS
LIN {X -112.139,Y -15.970,Z -37.437,A -90.000,B 90.000,C 0.000} C_DIS
LIN {X -112.068,Y -15.978,Z -37.265,A -90.000,B 90.000,C 0.000} C_DIS
LIN {X -112.019,Y -15.984,Z -37.149,A -90.000,B 90.000,C 0.000} C_DIS
LIN {X -111.905,Y -16.000,Z -36.895,A -90.000,B 90.000,C 0.000} C_DIS
LIN {X -111.774,Y -16.006,Z -36.642,A -90.000,B 90.000,C 0.000} C_DIS
LIN {X -111.574,Y -16.025,Z -36.299,A -90.000,B 90.000,C 0.000} C_DIS
LIN {X -111.544,Y -16.026,Z -36.250,A -90.000,B 90.000,C 0.000} C_DIS
LIN {X -111.460,Y -16.027,Z -36.127,A -90.000,B 90.000,C 0.000} C_DIS
LIN {X -111.306,Y -16.035,Z -35.914,A -90.000,B 90.000,C 0.000} C_DIS
LIN {X -111.172,Y -16.045,Z -35.738,A -90.000,B 90.000,C 0.000} C_DIS
LIN {X -111.017,Y -16.044,Z -35.556,A -90.000,B 90.000,C 0.000} C_DIS
LIN {X -110.916,Y -16.046,Z -35.446,A -90.000,B 90.000,C 0.000} C_DIS
LIN {X -110.692,Y -16.060,Z -35.225,A -90.000,B 90.000,C 0.000} C_DIS
LIN {X -110.372,Y -16.059,Z -34.940,A -90.000,B 90.000,C 0.000} C_DIS
LIN {X -110.280,Y -16.056,Z -34.866,A -90.000,B 90.000,C 0.000} C_DIS
LIN {X -110.132,Y -16.058,Z -34.759,A -90.000,B 90.000,C 0.000} C_DIS
LIN {X -109.941,Y -16.060,Z -34.626,A -90.000,B 90.000,C 0.000} C_DIS
LIN {X -109.825,Y -16.061,Z -34.548,A -90.000,B 90.000,C 0.000} C_DIS
LIN {X -109.574,Y -16.075,Z -34.395,A -90.000,B 90.000,C 0.000} C_DIS
LIN {X -109.476,Y -16.087,Z -34.330,A -90.000,B 90.000,C 0.000} C_DIS
LIN {X -109.153,Y -16.160,Z -34.105,A -90.000,B 90.000,C 0.000} C_DIS
LIN {X -109.026,Y -16.193,Z -34.022,A -90.000,B 90.000,C 0.000} C_DIS
LIN {X -108.874,Y -16.188,Z -33.822,A -90.000,B 90.000,C 0.000} C_DIS
LIN {X -108.791,Y -16.189,Z -33.712,A -90.000,B 90.000,C 0.000} C_DIS
LIN {X -108.649,Y -16.184,Z -33.533,A -90.000,B 90.000,C 0.000} C_DIS
LIN {X -108.470,Y -16.184,Z -33.324,A -90.000,B 90.000,C 0.000} C_DIS
LIN {X -108.289,Y -16.180,Z -33.106,A -90.000,B 90.000,C 0.000} C_DIS
LIN {X -108.197,Y -16.181,Z -32.998,A -90.000,B 90.000,C 0.000} C_DIS
LIN {X -108.115,Y -16.180,Z -32.918,A -90.000,B 90.000,C 0.000} C_DIS
LIN {X -107.776,Y -16.178,Z -32.589,A -90.000,B 90.000,C 0.000} C_DIS
LIN {X -107.568,Y -16.175,Z -32.393,A -90.000,B 90.000,C 0.000} C_DIS
LIN {X -107.420,Y -16.171,Z -32.258,A -90.000,B 90.000,C 0.000} C_DIS
LIN {X -107.332,Y -16.170,Z -32.182,A -90.000,B 90.000,C 0.000} C_DIS
LIN {X -107.031,Y -16.174,Z -31.933,A -90.000,B 90.000,C 0.000} C_DIS
LIN {X -106.682,Y -16.170,Z -31.658,A -90.000,B 90.000,C 0.000} C_DIS
LIN {X -106.534,Y -16.173,Z -31.547,A -90.000,B 90.000,C 0.000} C_DIS
LIN {X -105.950,Y -16.177,Z -31.118,A -90.000,B 90.000,C 0.000} C_DIS
LIN {X -105.711,Y -16.183,Z -30.951,A -90.000,B 90.000,C 0.000} C_DIS
LIN {X -105.348,Y -16.188,Z -30.703,A -90.000,B 90.000,C 0.000} C_DIS
LIN {X -104.976,Y -16.187,Z -30.453,A -90.000,B 90.000,C 0.000} C_DIS
LIN {X -104.724,Y -16.188,Z -30.289,A -90.000,B 90.000,C 0.000} C_DIS
LIN {X -104.320,Y -16.177,Z -30.046,A -90.000,B 90.000,C 0.000} C_DIS
LIN {X -104.185,Y -16.175,Z -29.967,A -90.000,B 90.000,C 0.000} C_DIS
LIN {X -103.829,Y -16.171,Z -29.777,A -90.000,B 90.000,C 0.000} C_DIS
LIN {X -103.608,Y -16.160,Z -29.666,A -90.000,B 90.000,C 0.000} C_DIS
LIN {X -103.294,Y -16.148,Z -29.508,A -90.000,B 90.000,C 0.000} C_DIS
LIN {X -103.218,Y -16.147,Z -29.470,A -90.000,B 90.000,C 0.000} C_DIS
LIN {X -103.042,Y -16.136,Z -29.393,A -90.000,B 90.000,C 0.000} C_DIS
LIN {X -102.947,Y -16.132,Z -29.353,A -90.000,B 90.000,C 0.000} C_DIS
LIN {X -102.731,Y -16.121,Z -29.266,A -90.000,B 90.000,C 0.000} C_DIS
LIN {X -102.524,Y -16.112,Z -29.182,A -90.000,B 90.000,C 0.000} C_DIS
LIN {X -102.239,Y -16.106,Z -29.072,A -90.000,B 90.000,C 0.000} C_DIS
LIN {X -101.799,Y -16.098,Z -28.912,A -90.000,B 90.000,C 0.000} C_DIS
LIN {X -101.734,Y -16.057,Z -28.837,A -90.000,B 90.000,C 0.000} C_DIS
LIN {X -101.593,Y -15.981,Z -28.684,A -90.000,B 90.000,C 0.000} C_DIS
LIN {X -101.501,Y -15.987,Z -28.480,A -90.000,B 90.000,C 0.000} C_DIS
LIN {X -101.459,Y -15.989,Z -28.391,A -90.000,B 90.000,C 0.000} C_DIS
LIN {X -101.274,Y -15.987,Z -28.028,A -90.000,B 90.000,C 0.000} C_DIS
LIN {X -101.231,Y -15.983,Z -27.955,A -90.000,B 90.000,C 0.000} C_DIS
LIN {X -101.029,Y -15.980,Z -27.636,A -90.000,B 90.000,C 0.000} C_DIS
LIN {X -100.795,Y -15.973,Z -27.281,A -90.000,B 90.000,C 0.000} C_DIS
LIN {X -100.631,Y -15.970,Z -27.041,A -90.000,B 90.000,C 0.000} C_DIS
LIN {X -100.431,Y -15.976,Z -26.770,A -90.000,B 90.000,C 0.000} C_DIS
LIN {X -100.274,Y -15.973,Z -26.570,A -90.000,B 90.000,C 0.000} C_DIS
LIN {X -100.120,Y -15.974,Z -26.381,A -90.000,B 90.000,C 0.000} C_DIS
LIN {X -99.730,Y -15.968,Z -25.928,A -90.000,B 90.000,C 0.000} C_DIS
LIN {X -99.517,Y -15.967,Z -25.689,A -90.000,B 90.000,C 0.000} C_DIS
LIN {X -99.406,Y -15.963,Z -25.571,A -90.000,B 90.000,C 0.000} C_DIS
LIN {X -99.247,Y -15.964,Z -25.401,A -90.000,B 90.000,C 0.000} C_DIS
LIN {X -99.007,Y -15.957,Z -25.166,A -90.000,B 90.000,C 0.000} C_DIS
LIN {X -98.882,Y -15.952,Z -25.049,A -90.000,B 90.000,C 0.000} C_DIS
LIN {X -98.711,Y -15.948,Z -24.892,A -90.000,B 90.000,C 0.000} C_DIS
LIN {X -98.487,Y -15.940,Z -24.695,A -90.000,B 90.000,C 0.000} C_DIS
LIN {X -98.384,Y -15.931,Z -24.607,A -90.000,B 90.000,C 0.000} C_DIS
LIN {X -98.061,Y -15.913,Z -24.343,A -90.000,B 90.000,C 0.000} C_DIS
LIN {X -97.977,Y -15.907,Z -24.277,A -90.000,B 90.000,C 0.000} C_DIS
LIN {X -97.742,Y -15.902,Z -24.106,A -90.000,B 90.000,C 0.000} C_DIS
LIN {X -97.564,Y -15.893,Z -23.992,A -90.000,B 90.000,C 0.000} C_DIS
LIN {X -97.509,Y -15.892,Z -23.956,A -90.000,B 90.000,C 0.000} C_DIS
LIN {X -97.427,Y -15.887,Z -23.905,A -90.000,B 90.000,C 0.000} C_DIS
LIN {X -97.263,Y -15.878,Z -23.807,A -90.000,B 90.000,C 0.000} C_DIS
LIN {X -97.146,Y -15.878,Z -23.744,A -90.000,B 90.000,C 0.000} C_DIS
LIN {X -96.765,Y -15.857,Z -23.573,A -90.000,B 90.000,C 0.000} C_DIS
LIN {X -96.659,Y -15.849,Z -23.538,A -90.000,B 90.000,C 0.000} C_DIS
LIN {X -96.267,Y -15.830,Z -23.416,A -90.000,B 90.000,C 0.000} C_DIS
LIN {X -96.136,Y -15.823,Z -23.376,A -90.000,B 90.000,C 0.000} C_DIS
LIN {X -96.018,Y -15.812,Z -23.346,A -90.000,B 90.000,C 0.000} C_DIS
LIN {X -95.723,Y -15.798,Z -23.282,A -90.000,B 90.000,C 0.000} C_DIS
LIN {X -95.458,Y -15.776,Z -23.247,A -90.000,B 90.000,C 0.000} C_DIS
LIN {X -95.301,Y -15.767,Z -23.228,A -90.000,B 90.000,C 0.000} C_DIS
LIN {X -94.883,Y -15.727,Z -23.219,A -90.000,B 90.000,C 0.000} C_DIS
LIN {X -94.746,Y -15.711,Z -23.223,A -90.000,B 90.000,C 0.000} C_DIS
LIN {X -94.557,Y -15.698,Z -23.236,A -90.000,B 90.000,C 0.000} C_DIS
LIN {X -94.197,Y -15.672,Z -23.265,A -90.000,B 90.000,C 0.000} C_DIS
LIN {X -93.771,Y -15.640,Z -23.331,A -90.000,B 90.000,C 0.000} C_DIS
LIN {X -93.310,Y -15.583,Z -23.442,A -90.000,B 90.000,C 0.000} C_DIS
LIN {X -92.899,Y -15.543,Z -23.568,A -90.000,B 90.000,C 0.000} C_DIS
LIN {X -92.621,Y -15.504,Z -23.679,A -90.000,B 90.000,C 0.000} C_DIS
LIN {X -92.505,Y -15.491,Z -23.725,A -90.000,B 90.000,C 0.000} C_DIS
LIN {X -92.309,Y -15.473,Z -23.806,A -90.000,B 90.000,C 0.000} C_DIS
LIN {X -92.241,Y -15.465,Z -23.837,A -90.000,B 90.000,C 0.000} C_DIS
LIN {X -91.949,Y -15.425,Z -23.973,A -90.000,B 90.000,C 0.000} C_DIS
LIN {X -91.683,Y -15.398,Z -24.084,A -90.000,B 90.000,C 0.000} C_DIS
LIN {X -91.379,Y -15.364,Z -24.236,A -90.000,B 90.000,C 0.000} C_DIS
LIN {X -91.098,Y -15.343,Z -24.352,A -90.000,B 90.000,C 0.000} C_DIS
LIN {X -90.920,Y -15.334,Z -24.411,A -90.000,B 90.000,C 0.000} C_DIS
LIN {X -90.600,Y -15.324,Z -24.488,A -90.000,B 90.000,C 0.000} C_DIS
LIN {X -90.256,Y -15.318,Z -24.537,A -90.000,B 90.000,C 0.000} C_DIS
LIN {X -90.167,Y -15.317,Z -24.550,A -90.000,B 90.000,C 0.000} C_DIS
LIN {X -89.774,Y -15.313,Z -24.578,A -90.000,B 90.000,C 0.000} C_DIS
LIN {X -89.305,Y -15.310,Z -24.582,A -90.000,B 90.000,C 0.000} C_DIS
LIN {X -89.048,Y -15.309,Z -24.566,A -90.000,B 90.000,C 0.000} C_DIS
LIN {X -89.200,Y -15.312,Z -24.520,A -90.000,B 90.000,C 0.000} C_DIS
LIN {X -89.349,Y -15.319,Z -24.469,A -90.000,B 90.000,C 0.000} C_DIS
LIN {X -89.495,Y -15.328,Z -24.414,A -90.000,B 90.000,C 0.000} C_DIS
LIN {X -89.591,Y -15.336,Z -24.374,A -90.000,B 90.000,C 0.000} C_DIS
LIN {X -89.797,Y -15.355,Z -24.282,A -90.000,B 90.000,C 0.000} C_DIS
LIN {X -89.852,Y -15.362,Z -24.255,A -90.000,B 90.000,C 0.000} C_DIS
LIN {X -89.961,Y -15.379,Z -24.193,A -90.000,B 90.000,C 0.000} C_DIS
LIN {X -89.978,Y -15.387,Z -24.168,A -90.000,B 90.000,C 0.000} C_DIS
LIN {X -89.998,Y -15.399,Z -24.129,A -90.000,B 90.000,C 0.000} C_DIS
LIN {X -90.022,Y -15.435,Z -24.024,A -90.000,B 90.000,C 0.000} C_DIS
LIN {X -90.014,Y -15.470,Z -23.936,A -90.000,B 90.000,C 0.000} C_DIS
LIN {X -89.972,Y -15.512,Z -23.842,A -90.000,B 90.000,C 0.000} C_DIS
LIN {X -89.947,Y -15.530,Z -23.806,A -90.000,B 90.000,C 0.000} C_DIS
LIN {X -89.894,Y -15.561,Z -23.744,A -90.000,B 90.000,C 0.000} C_DIS
LIN {X -89.813,Y -15.595,Z -23.682,A -90.000,B 90.000,C 0.000} C_DIS
LIN {X -89.665,Y -15.634,Z -23.611,A -90.000,B 90.000,C 0.000} C_DIS
LIN {X -89.552,Y -15.667,Z -23.549,A -90.000,B 90.000,C 0.000} C_DIS
LIN {X -89.483,Y -15.686,Z -23.514,A -90.000,B 90.000,C 0.000} C_DIS
LIN {X -89.224,Y -15.761,Z -23.367,A -90.000,B 90.000,C 0.000} C_DIS
LIN {X -88.941,Y -15.839,Z -23.226,A -90.000,B 90.000,C 0.000} C_DIS
LIN {X -88.879,Y -15.854,Z -23.198,A -90.000,B 90.000,C 0.000} C_DIS
LIN {X -88.802,Y -15.866,Z -23.166,A -90.000,B 90.000,C 0.000} C_DIS
LIN {X -88.686,Y -15.886,Z -23.108,A -90.000,B 90.000,C 0.000} C_DIS
LIN {X -88.535,Y -15.906,Z -23.040,A -90.000,B 90.000,C 0.000} C_DIS
LIN {X -88.350,Y -15.929,Z -22.944,A -90.000,B 90.000,C 0.000} C_DIS
LIN {X -88.175,Y -15.952,Z -22.833,A -90.000,B 90.000,C 0.000} C_DIS
LIN {X -88.140,Y -15.958,Z -22.805,A -90.000,B 90.000,C 0.000} C_DIS
LIN {X -88.055,Y -15.985,Z -22.661,A -90.000,B 90.000,C 0.000} C_DIS
LIN {X -88.003,Y -16.000,Z -22.575,A -90.000,B 90.000,C 0.000} C_DIS
LIN {X -87.710,Y -16.045,Z -22.095,A -90.000,B 90.000,C 0.000} C_DIS
LIN {X -87.624,Y -16.048,Z -21.970,A -90.000,B 90.000,C 0.000} C_DIS
LIN {X -87.496,Y -16.047,Z -21.791,A -90.000,B 90.000,C 0.000} C_DIS
LIN {X -87.261,Y -16.024,Z -21.501,A -90.000,B 90.000,C 0.000} C_DIS
LIN {X -87.127,Y -16.007,Z -21.341,A -90.000,B 90.000,C 0.000} C_DIS
LIN {X -87.054,Y -15.992,Z -21.267,A -90.000,B 90.000,C 0.000} C_DIS
LIN {X -86.802,Y -15.928,Z -21.023,A -90.000,B 90.000,C 0.000} C_DIS
LIN {X -86.781,Y -15.923,Z -21.003,A -90.000,B 90.000,C 0.000} C_DIS
LIN {X -86.739,Y -15.902,Z -20.908,A -90.000,B 90.000,C 0.000} C_DIS
LIN {X -86.677,Y -15.873,Z -20.783,A -90.000,B 90.000,C 0.000} C_DIS
LIN {X -86.616,Y -15.840,Z -20.689,A -90.000,B 90.000,C 0.000} C_DIS
LIN {X -86.486,Y -15.773,Z -20.504,A -90.000,B 90.000,C 0.000} C_DIS
LIN {X -86.407,Y -15.734,Z -20.399,A -90.000,B 90.000,C 0.000} C_DIS
LIN {X -86.330,Y -15.696,Z -20.305,A -90.000,B 90.000,C 0.000} C_DIS
LIN {X -86.258,Y -15.659,Z -20.241,A -90.000,B 90.000,C 0.000} C_DIS
LIN {X -86.183,Y -15.624,Z -20.184,A -90.000,B 90.000,C 0.000} C_DIS
LIN {X -86.073,Y -15.577,Z -20.111,A -90.000,B 90.000,C 0.000} C_DIS
LIN {X -86.002,Y -15.548,Z -20.069,A -90.000,B 90.000,C 0.000} C_DIS
LIN {X -85.896,Y -15.508,Z -20.013,A -90.000,B 90.000,C 0.000} C_DIS
LIN {X -85.724,Y -15.448,Z -19.940,A -90.000,B 90.000,C 0.000} C_DIS
LIN {X -85.693,Y -15.460,Z -19.782,A -90.000,B 90.000,C 0.000} C_DIS
LIN {X -85.672,Y -15.464,Z -19.701,A -90.000,B 90.000,C 0.000} C_DIS
LIN {X -85.656,Y -15.470,Z -19.619,A -90.000,B 90.000,C 0.000} C_DIS
LIN {X -85.620,Y -15.476,Z -19.493,A -90.000,B 90.000,C 0.000} C_DIS
LIN {X -85.529,Y -15.498,Z -19.197,A -90.000,B 90.000,C 0.000} C_DIS
LIN {X -85.482,Y -15.504,Z -19.072,A -90.000,B 90.000,C 0.000} C_DIS
LIN {X -85.424,Y -15.511,Z -18.933,A -90.000,B 90.000,C 0.000} C_DIS
LIN {X -85.248,Y -15.536,Z -18.523,A -90.000,B 90.000,C 0.000} C_DIS
LIN {X -85.191,Y -15.541,Z -18.418,A -90.000,B 90.000,C 0.000} C_DIS
LIN {X -85.031,Y -15.559,Z -18.140,A -90.000,B 90.000,C 0.000} C_DIS
LIN {X -85.001,Y -15.561,Z -18.093,A -90.000,B 90.000,C 0.000} C_DIS
LIN {X -84.863,Y -15.565,Z -17.890,A -90.000,B 90.000,C 0.000} C_DIS
LIN {X -84.731,Y -15.571,Z -17.702,A -90.000,B 90.000,C 0.000} C_DIS
LIN {X -84.594,Y -15.583,Z -17.516,A -90.000,B 90.000,C 0.000} C_DIS
LIN {X -84.408,Y -15.586,Z -17.302,A -90.000,B 90.000,C 0.000} C_DIS
LIN {X -84.302,Y -15.593,Z -17.184,A -90.000,B 90.000,C 0.000} C_DIS
LIN {X -84.230,Y -15.595,Z -17.116,A -90.000,B 90.000,C 0.000} C_DIS
LIN {X -84.045,Y -15.598,Z -16.944,A -90.000,B 90.000,C 0.000} C_DIS
LIN {X -83.711,Y -15.606,Z -16.639,A -90.000,B 90.000,C 0.000} C_DIS
LIN {X -83.452,Y -15.603,Z -16.444,A -90.000,B 90.000,C 0.000} C_DIS
LIN {X -83.359,Y -15.604,Z -16.376,A -90.000,B 90.000,C 0.000} C_DIS
LIN {X -83.005,Y -15.603,Z -16.153,A -90.000,B 90.000,C 0.000} C_DIS
LIN {X -82.629,Y -15.599,Z -15.932,A -90.000,B 90.000,C 0.000} C_DIS
LIN {X -82.598,Y -15.598,Z -15.915,A -90.000,B 90.000,C 0.000} C_DIS
LIN {X -82.266,Y -15.594,Z -15.754,A -90.000,B 90.000,C 0.000} C_DIS
LIN {X -82.109,Y -15.589,Z -15.686,A -90.000,B 90.000,C 0.000} C_DIS
LIN {X -81.831,Y -15.589,Z -15.570,A -90.000,B 90.000,C 0.000} C_DIS
LIN {X -81.623,Y -15.587,Z -15.491,A -90.000,B 90.000,C 0.000} C_DIS
LIN {X -81.385,Y -15.587,Z -15.405,A -90.000,B 90.000,C 0.000} C_DIS
LIN {X -81.073,Y -15.573,Z -15.317,A -90.000,B 90.000,C 0.000} C_DIS
LIN {X -80.962,Y -15.573,Z -15.289,A -90.000,B 90.000,C 0.000} C_DIS
LIN {X -80.384,Y -15.574,Z -15.146,A -90.000,B 90.000,C 0.000} C_DIS
LIN {X -80.163,Y -15.565,Z -15.111,A -90.000,B 90.000,C 0.000} C_DIS
LIN {X -79.960,Y -15.558,Z -15.080,A -90.000,B 90.000,C 0.000} C_DIS
LIN {X -79.438,Y -15.558,Z -15.009,A -90.000,B 90.000,C 0.000} C_DIS
LIN {X -79.240,Y -15.561,Z -14.985,A -90.000,B 90.000,C 0.000} C_DIS
LIN {X -79.163,Y -15.561,Z -14.977,A -90.000,B 90.000,C 0.000} C_DIS
LIN {X -78.685,Y -15.551,Z -14.959,A -90.000,B 90.000,C 0.000} C_DIS
LIN {X -78.181,Y -15.550,Z -14.949,A -90.000,B 90.000,C 0.000} C_DIS
LIN {X -77.902,Y -15.556,Z -14.947,A -90.000,B 90.000,C 0.000} C_DIS
LIN {X -77.603,Y -15.558,Z -14.954,A -90.000,B 90.000,C 0.000} C_DIS
LIN {X -77.465,Y -15.555,Z -14.964,A -90.000,B 90.000,C 0.000} C_DIS
LIN {X -77.248,Y -15.549,Z -14.985,A -90.000,B 90.000,C 0.000} C_DIS
LIN {X -76.825,Y -15.545,Z -15.031,A -90.000,B 90.000,C 0.000} C_DIS
LIN {X -76.773,Y -15.545,Z -15.037,A -90.000,B 90.000,C 0.000} C_DIS
LIN {X -76.321,Y -15.556,Z -15.099,A -90.000,B 90.000,C 0.000} C_DIS
LIN {X -75.946,Y -15.561,Z -15.158,A -90.000,B 90.000,C 0.000} C_DIS
LIN {X -75.514,Y -15.552,Z -15.256,A -90.000,B 90.000,C 0.000} C_DIS
LIN {X -75.267,Y -15.550,Z -15.316,A -90.000,B 90.000,C 0.000} C_DIS
LIN {X -74.846,Y -15.556,Z -15.429,A -90.000,B 90.000,C 0.000} C_DIS
LIN {X -74.562,Y -15.560,Z -15.509,A -90.000,B 90.000,C 0.000} C_DIS
LIN {X -74.278,Y -15.560,Z -15.594,A -90.000,B 90.000,C 0.000} C_DIS
LIN {X -73.839,Y -15.553,Z -15.746,A -90.000,B 90.000,C 0.000} C_DIS
LIN {X -73.684,Y -15.549,Z -15.802,A -90.000,B 90.000,C 0.000} C_DIS
LIN {X -73.601,Y -15.549,Z -15.833,A -90.000,B 90.000,C 0.000} C_DIS
LIN {X -72.899,Y -15.562,Z -16.103,A -90.000,B 90.000,C 0.000} C_DIS
LIN {X -72.552,Y -15.568,Z -16.239,A -90.000,B 90.000,C 0.000} C_DIS
LIN {X -72.378,Y -15.567,Z -16.315,A -90.000,B 90.000,C 0.000} C_DIS
LIN {X -72.129,Y -15.562,Z -16.432,A -90.000,B 90.000,C 0.000} C_DIS
LIN {X -71.421,Y -15.573,Z -16.791,A -90.000,B 90.000,C 0.000} C_DIS
LIN {X -70.952,Y -15.577,Z -17.035,A -90.000,B 90.000,C 0.000} C_DIS
LIN {X -70.767,Y -15.580,Z -17.127,A -90.000,B 90.000,C 0.000} C_DIS
LIN {X -70.379,Y -15.577,Z -17.342,A -90.000,B 90.000,C 0.000} C_DIS
LIN {X -69.856,Y -15.584,Z -17.639,A -90.000,B 90.000,C 0.000} C_DIS
LIN {X -69.178,Y -15.596,Z -18.015,A -90.000,B 90.000,C 0.000} C_DIS
LIN {X -68.983,Y -15.596,Z -18.129,A -90.000,B 90.000,C 0.000} C_DIS
LIN {X -68.523,Y -15.606,Z -18.404,A -90.000,B 90.000,C 0.000} C_DIS
LIN {X -67.562,Y -15.647,Z -18.992,A -90.000,B 90.000,C 0.000} C_DIS
LIN {X -67.302,Y -15.651,Z -19.165,A -90.000,B 90.000,C 0.000} C_DIS
LIN {X -67.021,Y -15.661,Z -19.358,A -90.000,B 90.000,C 0.000} C_DIS
LIN {X -66.472,Y -15.687,Z -19.739,A -90.000,B 90.000,C 0.000} C_DIS
LIN {X -66.275,Y -15.695,Z -19.879,A -90.000,B 90.000,C 0.000} C_DIS
LIN {X -65.998,Y -15.709,Z -20.082,A -90.000,B 90.000,C 0.000} C_DIS
LIN {X -65.701,Y -15.725,Z -20.304,A -90.000,B 90.000,C 0.000} C_DIS
LIN {X -65.201,Y -15.759,Z -20.681,A -90.000,B 90.000,C 0.000} C_DIS
LIN {X -65.130,Y -15.760,Z -20.740,A -90.000,B 90.000,C 0.000} C_DIS
LIN {X -64.796,Y -15.783,Z -21.036,A -90.000,B 90.000,C 0.000} C_DIS
LIN {X -64.299,Y -15.838,Z -21.451,A -90.000,B 90.000,C 0.000} C_DIS
LIN {X -63.992,Y -15.856,Z -21.722,A -90.000,B 90.000,C 0.000} C_DIS
LIN {X -63.883,Y -15.858,Z -21.824,A -90.000,B 90.000,C 0.000} C_DIS
LIN {X -63.785,Y -15.864,Z -21.920,A -90.000,B 90.000,C 0.000} C_DIS
LIN {X -63.695,Y -15.873,Z -22.012,A -90.000,B 90.000,C 0.000} C_DIS
LIN {X -63.628,Y -15.884,Z -22.075,A -90.000,B 90.000,C 0.000} C_DIS
LIN {X -63.217,Y -15.940,Z -22.481,A -90.000,B 90.000,C 0.000} C_DIS
LIN {X -62.770,Y -15.977,Z -22.961,A -90.000,B 90.000,C 0.000} C_DIS
LIN {X -62.615,Y -16.006,Z -23.116,A -90.000,B 90.000,C 0.000} C_DIS
LIN {X -62.242,Y -16.049,Z -23.533,A -90.000,B 90.000,C 0.000} C_DIS
LIN {X -62.102,Y -16.069,Z -23.696,A -90.000,B 90.000,C 0.000} C_DIS
LIN {X -61.997,Y -16.087,Z -23.822,A -90.000,B 90.000,C 0.000} C_DIS
LIN {X -61.921,Y -16.107,Z -23.908,A -90.000,B 90.000,C 0.000} C_DIS
LIN {X -61.693,Y -16.146,Z -24.152,A -90.000,B 90.000,C 0.000} C_DIS
LIN {X -61.534,Y -16.172,Z -24.326,A -90.000,B 90.000,C 0.000} C_DIS
LIN {X -61.301,Y -16.210,Z -24.591,A -90.000,B 90.000,C 0.000} C_DIS
LIN {X -61.285,Y -16.214,Z -24.607,A -90.000,B 90.000,C 0.000} C_DIS
LIN {X -61.145,Y -16.234,Z -24.728,A -90.000,B 90.000,C 0.000} C_DIS
LIN {X -60.976,Y -16.259,Z -24.873,A -90.000,B 90.000,C 0.000} C_DIS
LIN {X -60.636,Y -16.266,Z -25.093,A -90.000,B 90.000,C 0.000} C_DIS
LIN {X -60.520,Y -16.276,Z -25.162,A -90.000,B 90.000,C 0.000} C_DIS
LIN {X -59.716,Y -16.271,Z -25.516,A -90.000,B 90.000,C 0.000} C_DIS
LIN {X -59.612,Y -16.265,Z -25.553,A -90.000,B 90.000,C 0.000} C_DIS
LIN {X -58.373,Y -16.247,Z -25.960,A -90.000,B 90.000,C 0.000} C_DIS
LIN {X -58.289,Y -16.244,Z -25.984,A -90.000,B 90.000,C 0.000} C_DIS
LIN {X -57.910,Y -16.238,Z -26.089,A -90.000,B 90.000,C 0.000} C_DIS
LIN {X -56.490,Y -16.213,Z -26.483,A -90.000,B 90.000,C 0.000} C_DIS
LIN {X -56.280,Y -16.210,Z -26.533,A -90.000,B 90.000,C 0.000} C_DIS
LIN {X -55.273,Y -16.205,Z -26.795,A -90.000,B 90.000,C 0.000} C_DIS
LIN {X -54.822,Y -16.206,Z -26.910,A -90.000,B 90.000,C 0.000} C_DIS
LIN {X -54.209,Y -16.202,Z -27.059,A -90.000,B 90.000,C 0.000} C_DIS
LIN {X -53.844,Y -16.201,Z -27.142,A -90.000,B 90.000,C 0.000} C_DIS
LIN {X -53.626,Y -16.203,Z -27.190,A -90.000,B 90.000,C 0.000} C_DIS
LIN {X -52.718,Y -16.193,Z -27.363,A -90.000,B 90.000,C 0.000} C_DIS
LIN {X -52.414,Y -16.187,Z -27.424,A -90.000,B 90.000,C 0.000} C_DIS
LIN {X -51.927,Y -16.185,Z -27.532,A -90.000,B 90.000,C 0.000} C_DIS
LIN {X -51.576,Y -16.183,Z -27.602,A -90.000,B 90.000,C 0.000} C_DIS
LIN {X -50.654,Y -16.185,Z -27.777,A -90.000,B 90.000,C 0.000} C_DIS
LIN {X -50.438,Y -16.188,Z -27.816,A -90.000,B 90.000,C 0.000} C_DIS
LIN {X -48.937,Y -16.181,Z -28.036,A -90.000,B 90.000,C 0.000} C_DIS
LIN {X -48.704,Y -16.179,Z -28.061,A -90.000,B 90.000,C 0.000} C_DIS
LIN {X -45.499,Y -16.167,Z -28.442,A -90.000,B 90.000,C 0.000} C_DIS
LIN {X -45.375,Y -16.164,Z -28.453,A -90.000,B 90.000,C 0.000} C_DIS
LIN {X -45.093,Y -16.162,Z -28.477,A -90.000,B 90.000,C 0.000} C_DIS
LIN {X -43.884,Y -16.142,Z -28.598,A -90.000,B 90.000,C 0.000} C_DIS
LIN {X -41.817,Y -16.110,Z -28.819,A -90.000,B 90.000,C 0.000} C_DIS
LIN {X -40.562,Y -16.069,Z -28.950,A -90.000,B 90.000,C 0.000} C_DIS
LIN {X -40.040,Y -16.050,Z -29.006,A -90.000,B 90.000,C 0.000} C_DIS
LIN {X -39.052,Y -16.030,Z -29.140,A -90.000,B 90.000,C 0.000} C_DIS
LIN {X -37.630,Y -15.991,Z -29.351,A -90.000,B 90.000,C 0.000} C_DIS
LIN {X -37.224,Y -15.982,Z -29.410,A -90.000,B 90.000,C 0.000} C_DIS
LIN {X -36.832,Y -15.971,Z -29.469,A -90.000,B 90.000,C 0.000} C_DIS
LIN {X -35.961,Y -15.940,Z -29.607,A -90.000,B 90.000,C 0.000} C_DIS
LIN {X -35.295,Y -15.923,Z -29.720,A -90.000,B 90.000,C 0.000} C_DIS
LIN {X -34.851,Y -15.909,Z -29.798,A -90.000,B 90.000,C 0.000} C_DIS
LIN {X -34.212,Y -15.884,Z -29.916,A -90.000,B 90.000,C 0.000} C_DIS
LIN {X -34.051,Y -15.880,Z -29.949,A -90.000,B 90.000,C 0.000} C_DIS
LIN {X -31.415,Y -15.833,Z -30.472,A -90.000,B 90.000,C 0.000} C_DIS
LIN {X -29.754,Y -15.799,Z -30.804,A -90.000,B 90.000,C 0.000} C_DIS
LIN {X -29.050,Y -15.787,Z -30.948,A -90.000,B 90.000,C 0.000} C_DIS
LIN {X -27.877,Y -15.773,Z -31.182,A -90.000,B 90.000,C 0.000} C_DIS
LIN {X -27.355,Y -15.771,Z -31.290,A -90.000,B 90.000,C 0.000} C_DIS
LIN {X -27.056,Y -15.774,Z -31.346,A -90.000,B 90.000,C 0.000} C_DIS
LIN {X -26.172,Y -15.777,Z -31.509,A -90.000,B 90.000,C 0.000} C_DIS
LIN {X -25.108,Y -15.790,Z -31.696,A -90.000,B 90.000,C 0.000} C_DIS
LIN {X -24.686,Y -15.799,Z -31.765,A -90.000,B 90.000,C 0.000} C_DIS
LIN {X -23.940,Y -15.818,Z -31.876,A -90.000,B 90.000,C 0.000} C_DIS
LIN {X -23.715,Y -15.827,Z -31.906,A -90.000,B 90.000,C 0.000} C_DIS
LIN {X -23.219,Y -15.850,Z -31.976,A -90.000,B 90.000,C 0.000} C_DIS
LIN {X -22.370,Y -15.884,Z -32.105,A -90.000,B 90.000,C 0.000} C_DIS
LIN {X -21.459,Y -15.936,Z -32.233,A -90.000,B 90.000,C 0.000} C_DIS
LIN {X -20.866,Y -15.967,Z -32.320,A -90.000,B 90.000,C 0.000} C_DIS
LIN {X -20.521,Y -15.982,Z -32.374,A -90.000,B 90.000,C 0.000} C_DIS
LIN {X -20.237,Y -15.998,Z -32.418,A -90.000,B 90.000,C 0.000} C_DIS
LIN {X -19.534,Y -16.037,Z -32.528,A -90.000,B 90.000,C 0.000} C_DIS
LIN {X -18.548,Y -16.082,Z -32.683,A -90.000,B 90.000,C 0.000} C_DIS
LIN {X -18.287,Y -16.091,Z -32.720,A -90.000,B 90.000,C 0.000} C_DIS
LIN {X -17.724,Y -16.104,Z -32.805,A -90.000,B 90.000,C 0.000} C_DIS
LIN {X -17.252,Y -16.120,Z -32.888,A -90.000,B 90.000,C 0.000} C_DIS
LIN {X -15.931,Y -16.162,Z -33.129,A -90.000,B 90.000,C 0.000} C_DIS
LIN {X -15.588,Y -16.170,Z -33.187,A -90.000,B 90.000,C 0.000} C_DIS
LIN {X -14.914,Y -16.172,Z -33.310,A -90.000,B 90.000,C 0.000} C_DIS
LIN {X -14.450,Y -16.183,Z -33.407,A -90.000,B 90.000,C 0.000} C_DIS
LIN {X -14.238,Y -16.185,Z -33.449,A -90.000,B 90.000,C 0.000} C_DIS
LIN {X -12.656,Y -16.220,Z -33.740,A -90.000,B 90.000,C 0.000} C_DIS
LIN {X -12.343,Y -16.217,Z -33.789,A -90.000,B 90.000,C 0.000} C_DIS
LIN {X -11.271,Y -16.225,Z -33.982,A -90.000,B 90.000,C 0.000} C_DIS
LIN {X -10.979,Y -16.223,Z -34.028,A -90.000,B 90.000,C 0.000} C_DIS
LIN {X -10.792,Y -16.220,Z -34.059,A -90.000,B 90.000,C 0.000} C_DIS
LIN {X -10.130,Y -16.205,Z -34.172,A -90.000,B 90.000,C 0.000} C_DIS
LIN {X -10.045,Y -16.204,Z -34.188,A -90.000,B 90.000,C 0.000} C_DIS
LIN {X -9.657,Y -16.208,Z -34.257,A -90.000,B 90.000,C 0.000} C_DIS
LIN {X -9.327,Y -16.201,Z -34.310,A -90.000,B 90.000,C 0.000} C_DIS
LIN {X -8.174,Y -16.193,Z -34.517,A -90.000,B 90.000,C 0.000} C_DIS
LIN {X -7.899,Y -16.197,Z -34.563,A -90.000,B 90.000,C 0.000} C_DIS
LIN {X -6.805,Y -16.188,Z -34.706,A -90.000,B 90.000,C 0.000} C_DIS
LIN {X -6.494,Y -16.184,Z -34.748,A -90.000,B 90.000,C 0.000} C_DIS
LIN {X -6.394,Y -16.184,Z -34.761,A -90.000,B 90.000,C 0.000} C_DIS
LIN {X -6.169,Y -16.186,Z -34.793,A -90.000,B 90.000,C 0.000} C_DIS
LIN {X -5.813,Y -16.181,Z -34.831,A -90.000,B 90.000,C 0.000} C_DIS
LIN {X -5.714,Y -16.181,Z -34.844,A -90.000,B 90.000,C 0.000} C_DIS
LIN {X -5.107,Y -16.190,Z -34.935,A -90.000,B 90.000,C 0.000} C_DIS
LIN {X -4.098,Y -16.184,Z -35.101,A -90.000,B 90.000,C 0.000} C_DIS
LIN {X -3.649,Y -16.172,Z -35.165,A -90.000,B 90.000,C 0.000} C_DIS
LIN {X -3.107,Y -16.164,Z -35.228,A -90.000,B 90.000,C 0.000} C_DIS
LIN {X -2.407,Y -16.146,Z -35.313,A -90.000,B 90.000,C 0.000} C_DIS
LIN {X -1.937,Y -16.135,Z -35.370,A -90.000,B 90.000,C 0.000} C_DIS
LIN {X -1.032,Y -16.120,Z -35.489,A -90.000,B 90.000,C 0.000} C_DIS
LIN {X -0.883,Y -16.119,Z -35.507,A -90.000,B 90.000,C 0.000} C_DIS
LIN {X 0.671,Y -16.087,Z -35.664,A -90.000,B 90.000,C 0.000} C_DIS
LIN {X 1.010,Y -16.083,Z -35.702,A -90.000,B 90.000,C 0.000} C_DIS
LIN {X 1.661,Y -16.073,Z -35.778,A -90.000,B 90.000,C 0.000} C_DIS
LIN {X 2.644,Y -16.060,Z -35.891,A -90.000,B 90.000,C 0.000} C_DIS
LIN {X 3.300,Y -16.060,Z -35.978,A -90.000,B 90.000,C 0.000} C_DIS
LIN {X 4.217,Y -16.056,Z -36.103,A -90.000,B 90.000,C 0.000} C_DIS
LIN {X 4.728,Y -16.056,Z -36.181,A -90.000,B 90.000,C 0.000} C_DIS
